LIN {X 0,Y 509.842,Z 166.475,A -85,B 0,C 180,E1 -5630.648,E2 -5630.648} C_VEL
LIN {X 0,Y 509.826,Z 166.476,A -85,B 0,C 180,E1 -5633.734,E2 -5633.734} C_VEL
LIN {X 0,Y 509.16,Z 166.561,A -85,B 0,C 180,E1 -5634.394,E2 -5634.394} C_VEL
LIN {X 0,Y 506.343,Z 166.91,A -85,B 0,C 180,E1 -5635.466,E2 -5635.466} C_VEL
LIN {X 0,Y 503.95,Z 167.21,A -85,B 0,C 180,E1 -5636.329,E2 -5636.329} C_VEL
LIN {X 0,Y 502.902,Z 167.337,A -85,B 0,C 180,E1 -5636.996,E2 -5636.996} C_VEL
LIN {X 0,Y 502.805,Z 167.349,A -85,B 0,C 180,E1 -5637.221,E2 -5637.221} C_VEL
LIN {X 0,Y 502.826,Z 167.352,A -85,B 0,C 180,E1 -5640.062,E2 -5640.062} C_VEL
LIN {X 0,Y 502.83,Z 167.346,A -85,B 0,C 180,E1 -5642.533,E2 -5642.533} C_VEL
LIN {X 0,Y 502.824,Z 167.349,A -85,B 0,C 180,E1 -5645.299,E2 -5645.299} C_VEL
LIN {X 0,Y 502.781,Z 167.358,A -85,B 0,C 180,E1 -5647.827,E2 -5647.827} C_VEL
LIN {X 0,Y 502.821,Z 167.347,A -85,B 0,C 180,E1 -5650.4,E2 -5650.4} C_VEL
LIN {X 0,Y 502.83,Z 167.349,A -85,B 0,C 180,E1 -5652.932,E2 -5652.932} C_VEL
LIN {X 0,Y 502.848,Z 167.352,A -85,B 0,C 180,E1 -5655.43,E2 -5655.43} C_VEL
LIN {X 0,Y 502.874,Z 167.343,A -85,B 0,C 180,E1 -5658.717,E2 -5658.717} C_VEL
LIN {X 0,Y 502.899,Z 167.34,A -85,B 0,C 180,E1 -5661.967,E2 -5661.967} C_VEL
LIN {X 0,Y 502.939,Z 167.335,A -85,B 0,C 180,E1 -5664.387,E2 -5664.387} C_VEL
LIN {X 0,Y 503.023,Z 167.326,A -85,B 0,C 180,E1 -5667.598,E2 -5667.598} C_VEL
LIN {X 0,Y 503.025,Z 167.324,A -85,B 0,C 180,E1 -5670,E2 -5670} C_VEL
LIN {X 0,Y 503.023,Z 167.326,A -85,B 0,C 180,E1 -5672.402,E2 -5672.402} C_VEL
LIN {X 0,Y 502.939,Z 167.335,A -85,B 0,C 180,E1 -5675.613,E2 -5675.613} C_VEL
LIN {X 0,Y 502.899,Z 167.34,A -85,B 0,C 180,E1 -5678.033,E2 -5678.033} C_VEL
LIN {X 0,Y 502.874,Z 167.343,A -85,B 0,C 180,E1 -5681.283,E2 -5681.283} C_VEL
LIN {X 0,Y 502.848,Z 167.352,A -85,B 0,C 180,E1 -5684.57,E2 -5684.57} C_VEL
LIN {X 0,Y 502.858,Z 167.346,A -85,B 0,C 180,E1 -5687.907,E2 -5687.907} C_VEL
LIN {X 0,Y 502.824,Z 167.353,A -85,B 0,C 180,E1 -5690.536,E2 -5690.536} C_VEL
LIN {X 0,Y 502.793,Z 167.351,A -85,B 0,C 180,E1 -5693.04,E2 -5693.04} C_VEL
LIN {X 0,Y 502.836,Z 167.346,A -85,B 0,C 180,E1 -5695.675,E2 -5695.675} C_VEL
LIN {X 0,Y 502.838,Z 167.35,A -85,B 0,C 180,E1 -5698.372,E2 -5698.372} C_VEL
LIN {X 0,Y 502.792,Z 167.352,A -85,B 0,C 180,E1 -5701.5,E2 -5701.5} C_VEL
LIN {X 0,Y 502.801,Z 167.352,A -85,B 0,C 180,E1 -5704.445,E2 -5704.445} C_VEL
LIN {X 0,Y 502.776,Z 167.353,A -85,B 0,C 180,E1 -5707.178,E2 -5707.178} C_VEL
LIN {X 0,Y 502.816,Z 167.353,A -85,B 0,C 180,E1 -5710.012,E2 -5710.012} C_VEL
LIN {X 0,Y 502.767,Z 167.356,A -85,B 0,C 180,E1 -5713.231,E2 -5713.231} C_VEL
LIN {X 0,Y 502.784,Z 167.36,A -85,B 0,C 180,E1 -5715.661,E2 -5715.661} C_VEL
LIN {X 0,Y 502.82,Z 167.349,A -85,B 0,C 180,E1 -5719.004,E2 -5719.004} C_VEL
LIN {X 0,Y 502.788,Z 167.352,A -85,B 0,C 180,E1 -5722.046,E2 -5722.046} C_VEL
LIN {X 0,Y 502.803,Z 167.353,A -85,B 0,C 180,E1 -5725.035,E2 -5725.035} C_VEL
LIN {X 0,Y 502.778,Z 167.353,A -85,B 0,C 180,E1 -5727.916,E2 -5727.916} C_VEL
LIN {X 0,Y 502.833,Z 167.348,A -85,B 0,C 180,E1 -5730.713,E2 -5730.713} C_VEL
LIN {X 0,Y 502.855,Z 167.346,A -85,B 0,C 180,E1 -5733.439,E2 -5733.439} C_VEL
LIN {X 0,Y 502.784,Z 167.351,A -85,B 0,C 180,E1 -5736.086,E2 -5736.086} C_VEL
LIN {X 0,Y 502.777,Z 167.357,A -85,B 0,C 180,E1 -5738.689,E2 -5738.689} C_VEL
LIN {X 0,Y 502.823,Z 167.35,A -85,B 0,C 180,E1 -5741.249,E2 -5741.249} C_VEL
LIN {X 0,Y 502.816,Z 167.347,A -85,B 0,C 180,E1 -5743.767,E2 -5743.767} C_VEL
LIN {X 0,Y 502.825,Z 167.349,A -85,B 0,C 180,E1 -5746.255,E2 -5746.255} C_VEL
LIN {X 0,Y 502.87,Z 167.348,A -85,B 0,C 180,E1 -5748.717,E2 -5748.717} C_VEL
LIN {X 0,Y 502.895,Z 167.339,A -85,B 0,C 180,E1 -5751.967,E2 -5751.967} C_VEL
LIN {X 0,Y 502.931,Z 167.34,A -85,B 0,C 180,E1 -5754.387,E2 -5754.387} C_VEL
LIN {X 0,Y 503.017,Z 167.323,A -85,B 0,C 180,E1 -5757.598,E2 -5757.598} C_VEL
LIN {X 0,Y 503.019,Z 167.326,A -85,B 0,C 180,E1 -5760,E2 -5760} C_VEL
LIN {X 0,Y 503.017,Z 167.329,A -85,B 0,C 180,E1 -5762.403,E2 -5762.403} C_VEL
LIN {X 0,Y 502.929,Z 167.335,A -85,B 0,C 180,E1 -5765.614,E2 -5765.614} C_VEL
LIN {X 0,Y 502.896,Z 167.346,A -85,B 0,C 180,E1 -5768.034,E2 -5768.034} C_VEL
LIN {X 0,Y 502.872,Z 167.341,A -85,B 0,C 180,E1 -5771.284,E2 -5771.284} C_VEL
LIN {X 0,Y 502.84,Z 167.345,A -85,B 0,C 180,E1 -5774.571,E2 -5774.571} C_VEL
LIN {X 0,Y 502.85,Z 167.35,A -85,B 0,C 180,E1 -5777.908,E2 -5777.908} C_VEL
LIN {X 0,Y 502.824,Z 167.346,A -85,B 0,C 180,E1 -5780.537,E2 -5780.537} C_VEL
LIN {X 0,Y 502.789,Z 167.352,A -85,B 0,C 180,E1 -5783.041,E2 -5783.041} C_VEL
LIN {X 0,Y 502.835,Z 167.352,A -85,B 0,C 180,E1 -5785.676,E2 -5785.676} C_VEL
LIN {X 0,Y 502.833,Z 167.345,A -85,B 0,C 180,E1 -5788.374,E2 -5788.374} C_VEL
LIN {X 0,Y 502.789,Z 167.357,A -85,B 0,C 180,E1 -5791.499,E2 -5791.499} C_VEL
LIN {X 0,Y 502.8,Z 167.352,A -85,B 0,C 180,E1 -5793.995,E2 -5793.995} C_VEL
LIN {X 0,Y 502.775,Z 167.361,A -85,B 0,C 180,E1 -5797.178,E2 -5797.178} C_VEL
LIN {X 0,Y 502.785,Z 167.355,A -85,B 0,C 180,E1 -5800.016,E2 -5800.016} C_VEL
LIN {X 0,Y 502.801,Z 167.354,A -85,B 0,C 180,E1 -5802.2,E2 -5802.2} C_VEL
LIN {X 0,Y 502.757,Z 167.362,A -85,B 0,C 180,E1 -5803.374,E2 -5803.374} C_VEL
LIN {X 0,Y 502.897,Z 168.072,A -85,B 0,C 180,E1 -5804.544,E2 -5804.544} C_VEL
LIN {X 0,Y 503.501,Z 172.327,A -85,B 0,C 180,E1 -5807.714,E2 -5807.714} C_VEL
LIN {X 0,Y 503.568,Z 175.925,A -85,B 0,C 180,E1 -5810.14,E2 -5810.14} C_VEL
LIN {X 0,Y 503.28,Z 180.665,A -85,B 0,C 180,E1 -5813.097,E2 -5813.097} C_VEL
LIN {X 0,Y 503.059,Z 185.701,A -85,B 0,C 180,E1 -5816.026,E2 -5816.026} C_VEL
LIN {X 0,Y 502.876,Z 190.836,A -85,B 0,C 180,E1 -5818.863,E2 -5818.863} C_VEL
LIN {X 0,Y 502.695,Z 196.322,A -85,B 0,C 180,E1 -5821.737,E2 -5821.737} C_VEL
LIN {X 0,Y 502.576,Z 201.398,A -85,B 0,C 180,E1 -5824.31,E2 -5824.31} C_VEL
LIN {X 0,Y 502.48,Z 207.799,A -85,B 0,C 180,E1 -5827.387,E2 -5827.387} C_VEL
LIN {X 0,Y 502.354,Z 214.071,A -85,B 0,C 180,E1 -5830.381,E2 -5830.381} C_VEL
LIN {X 0,Y 502.241,Z 219.461,A -85,B 0,C 180,E1 -5832.911,E2 -5832.911} C_VEL
LIN {X 0,Y 502.211,Z 225.524,A -85,B 0,C 180,E1 -5835.721,E2 -5835.721} C_VEL
LIN {X 0,Y 504.275,Z 237.727,A -85,B 0,C 180,E1 -5836.089,E2 -5836.089} C_VEL
LIN {X 0,Y 504.627,Z 241.055,A -85,B 0,C 180,E1 -5836.202,E2 -5836.202} C_VEL
LIN {X 0,Y 504.312,Z 253.379,A -85,B 0,C 180,E1 -5836.707,E2 -5836.707} C_VEL
LIN {X 0,Y 504.006,Z 263.916,A -85,B 0,C 180,E1 -5837.276,E2 -5837.276} C_VEL
LIN {X 0,Y 503.684,Z 273.477,A -85,B 0,C 180,E1 -5837.919,E2 -5837.919} C_VEL
LIN {X 0,Y 503.425,Z 282.175,A -85,B 0,C 180,E1 -5838.627,E2 -5838.627} C_VEL
LIN {X 0,Y 503.194,Z 289.542,A -85,B 0,C 180,E1 -5839.336,E2 -5839.336} C_VEL
LIN {X 0,Y 502.944,Z 296.73,A -85,B 0,C 180,E1 -5840.144,E2 -5840.144} C_VEL
LIN {X 0,Y 502.683,Z 304.275,A -85,B 0,C 180,E1 -5841.153,E2 -5841.153} C_VEL
LIN {X 0,Y 502.471,Z 310.565,A -85,B 0,C 180,E1 -5842.162,E2 -5842.162} C_VEL
LIN {X 0,Y 502.317,Z 315.989,A -85,B 0,C 180,E1 -5843.21,E2 -5843.21} C_VEL
LIN {X 0,Y 502.256,Z 320.895,A -85,B 0,C 180,E1 -5844.379,E2 -5844.379} C_VEL
LIN {X 0,Y 502.128,Z 324.85,A -85,B 0,C 180,E1 -5845.585,E2 -5845.585} C_VEL
LIN {X 0,Y 502.122,Z 327.772,A -85,B 0,C 180,E1 -5846.791,E2 -5846.791} C_VEL
LIN {X 0,Y 502.036,Z 330.196,A -85,B 0,C 180,E1 -5848.396,E2 -5848.396} C_VEL
LIN {X 0,Y 501.99,Z 330.78,A -85,B 0,C 180,E1 -5849.198,E2 -5849.198} C_VEL
LIN {X 0,Y 501.99,Z 330.78,A -85,B 0,C 180,E1 -5850.802,E2 -5850.802} C_VEL
LIN {X 0,Y 502.036,Z 330.196,A -85,B 0,C 180,E1 -5851.604,E2 -5851.604} C_VEL
LIN {X 0,Y 502.122,Z 327.772,A -85,B 0,C 180,E1 -5853.209,E2 -5853.209} C_VEL
LIN {X 0,Y 502.128,Z 324.85,A -85,B 0,C 180,E1 -5854.415,E2 -5854.415} C_VEL
LIN {X 0,Y 502.257,Z 320.895,A -85,B 0,C 180,E1 -5855.621,E2 -5855.621} C_VEL
LIN {X 0,Y 502.317,Z 315.989,A -85,B 0,C 180,E1 -5856.79,E2 -5856.79} C_VEL
LIN {X 0,Y 502.471,Z 310.565,A -85,B 0,C 180,E1 -5857.838,E2 -5857.838} C_VEL
LIN {X 0,Y 502.683,Z 304.275,A -85,B 0,C 180,E1 -5858.847,E2 -5858.847} C_VEL
LIN {X 0,Y 502.944,Z 296.73,A -85,B 0,C 180,E1 -5859.856,E2 -5859.856} C_VEL
LIN {X 0,Y 503.237,Z 287.621,A -85,B 0,C 180,E1 -5860.867,E2 -5860.867} C_VEL
LIN {X 0,Y 503.648,Z 276.174,A -85,B 0,C 180,E1 -5861.878,E2 -5861.878} C_VEL
LIN {X 0,Y 503.876,Z 266.59,A -85,B 0,C 180,E1 -5862.559,E2 -5862.559} C_VEL
LIN {X 0,Y 504.174,Z 256.395,A -85,B 0,C 180,E1 -5863.143,E2 -5863.143} C_VEL
LIN {X 0,Y 504.477,Z 246.331,A -85,B 0,C 180,E1 -5863.597,E2 -5863.597} C_VEL
LIN {X 0,Y 504.441,Z 238.601,A -85,B 0,C 180,E1 -5863.88,E2 -5863.88} C_VEL
LIN {X 0,Y 502.532,Z 227.434,A -85,B 0,C 180,E1 -5864.227,E2 -5864.227} C_VEL
LIN {X 0,Y 502.211,Z 225.524,A -85,B 0,C 180,E1 -5864.279,E2 -5864.279} C_VEL
LIN {X 0,Y 502.241,Z 219.461,A -85,B 0,C 180,E1 -5867.089,E2 -5867.089} C_VEL
LIN {X 0,Y 502.421,Z 212.275,A -85,B 0,C 180,E1 -5870.469,E2 -5870.469} C_VEL
LIN {X 0,Y 502.479,Z 206.885,A -85,B 0,C 180,E1 -5873.055,E2 -5873.055} C_VEL
LIN {X 0,Y 502.576,Z 201.398,A -85,B 0,C 180,E1 -5875.69,E2 -5875.69} C_VEL
LIN {X 0,Y 502.702,Z 196.094,A -85,B 0,C 180,E1 -5878.381,E2 -5878.381} C_VEL
LIN {X 0,Y 502.876,Z 190.832,A -85,B 0,C 180,E1 -5881.137,E2 -5881.137} C_VEL
LIN {X 0,Y 503.052,Z 185.669,A -85,B 0,C 180,E1 -5883.974,E2 -5883.974} C_VEL
LIN {X 0,Y 503.329,Z 180.065,A -85,B 0,C 180,E1 -5887.26,E2 -5887.26} C_VEL
LIN {X 0,Y 503.544,Z 175.787,A -85,B 0,C 180,E1 -5889.942,E2 -5889.942} C_VEL
LIN {X 0,Y 503.509,Z 172.318,A -85,B 0,C 180,E1 -5892.287,E2 -5892.287} C_VEL
LIN {X 0,Y 502.897,Z 168.091,A -85,B 0,C 180,E1 -5895.456,E2 -5895.456} C_VEL
LIN {X 0,Y 502.755,Z 167.361,A -85,B 0,C 180,E1 -5896.766,E2 -5896.766} C_VEL
LIN {X 0,Y 502.796,Z 167.358,A -85,B 0,C 180,E1 -5899.007,E2 -5899.007} C_VEL
LIN {X 0,Y 502.79,Z 167.354,A -85,B 0,C 180,E1 -5902.045,E2 -5902.045} C_VEL
LIN {X 0,Y 502.795,Z 167.357,A -85,B 0,C 180,E1 -5905.033,E2 -5905.033} C_VEL
LIN {X 0,Y 502.78,Z 167.352,A -85,B 0,C 180,E1 -5907.915,E2 -5907.915} C_VEL
LIN {X 0,Y 502.818,Z 167.353,A -85,B 0,C 180,E1 -5910.711,E2 -5910.711} C_VEL
LIN {X 0,Y 502.859,Z 167.342,A -85,B 0,C 180,E1 -5913.439,E2 -5913.439} C_VEL
LIN {X 0,Y 502.787,Z 167.355,A -85,B 0,C 180,E1 -5916.086,E2 -5916.086} C_VEL
LIN {X 0,Y 502.779,Z 167.355,A -85,B 0,C 180,E1 -5918.688,E2 -5918.688} C_VEL
LIN {X 0,Y 502.824,Z 167.346,A -85,B 0,C 180,E1 -5921.248,E2 -5921.248} C_VEL
LIN {X 0,Y 502.816,Z 167.35,A -85,B 0,C 180,E1 -5923.767,E2 -5923.767} C_VEL
LIN {X 0,Y 502.825,Z 167.352,A -85,B 0,C 180,E1 -5926.254,E2 -5926.254} C_VEL
LIN {X 0,Y 502.872,Z 167.341,A -85,B 0,C 180,E1 -5928.716,E2 -5928.716} C_VEL
LIN {X 0,Y 502.896,Z 167.346,A -85,B 0,C 180,E1 -5931.966,E2 -5931.966} C_VEL
LIN {X 0,Y 502.929,Z 167.335,A -85,B 0,C 180,E1 -5934.386,E2 -5934.386} C_VEL
LIN {X 0,Y 503.017,Z 167.329,A -85,B 0,C 180,E1 -5937.597,E2 -5937.597} C_VEL
LIN {X 0,Y 503.019,Z 167.326,A -85,B 0,C 180,E1 -5940,E2 -5940} C_VEL
LIN {X 0,Y 503.017,Z 167.323,A -85,B 0,C 180,E1 -5942.402,E2 -5942.402} C_VEL
LIN {X 0,Y 502.931,Z 167.34,A -85,B 0,C 180,E1 -5945.613,E2 -5945.613} C_VEL
LIN {X 0,Y 502.895,Z 167.339,A -85,B 0,C 180,E1 -5948.033,E2 -5948.033} C_VEL
LIN {X 0,Y 502.87,Z 167.348,A -85,B 0,C 180,E1 -5951.283,E2 -5951.283} C_VEL
LIN {X 0,Y 502.838,Z 167.345,A -85,B 0,C 180,E1 -5954.571,E2 -5954.571} C_VEL
LIN {X 0,Y 502.855,Z 167.343,A -85,B 0,C 180,E1 -5957.907,E2 -5957.907} C_VEL
LIN {X 0,Y 502.822,Z 167.348,A -85,B 0,C 180,E1 -5960.536,E2 -5960.536} C_VEL
LIN {X 0,Y 502.787,Z 167.359,A -85,B 0,C 180,E1 -5963.04,E2 -5963.04} C_VEL
LIN {X 0,Y 502.833,Z 167.346,A -85,B 0,C 180,E1 -5965.675,E2 -5965.675} C_VEL
LIN {X 0,Y 502.836,Z 167.347,A -85,B 0,C 180,E1 -5968.372,E2 -5968.372} C_VEL
LIN {X 0,Y 502.787,Z 167.351,A -85,B 0,C 180,E1 -5971.499,E2 -5971.499} C_VEL
LIN {X 0,Y 502.8,Z 167.355,A -85,B 0,C 180,E1 -5974.445,E2 -5974.445} C_VEL
LIN {X 0,Y 502.774,Z 167.354,A -85,B 0,C 180,E1 -5977.178,E2 -5977.178} C_VEL
LIN {X 0,Y 502.815,Z 167.35,A -85,B 0,C 180,E1 -5980.012,E2 -5980.012} C_VEL
LIN {X 0,Y 502.767,Z 167.354,A -85,B 0,C 180,E1 -5983.231,E2 -5983.231} C_VEL
LIN {X 0,Y 502.783,Z 167.352,A -85,B 0,C 180,E1 -5985.661,E2 -5985.661} C_VEL
LIN {X 0,Y 502.813,Z 167.348,A -85,B 0,C 180,E1 -5989.005,E2 -5989.005} C_VEL
LIN {X 0,Y 502.789,Z 167.358,A -85,B 0,C 180,E1 -5992.046,E2 -5992.046} C_VEL
LIN {X 0,Y 502.805,Z 167.349,A -85,B 0,C 180,E1 -5995.035,E2 -5995.035} C_VEL
LIN {X 0,Y 502.805,Z 167.349,A -85,B 0,C 180,E1 -5997.221,E2 -5997.221} C_VEL
LIN {X 0,Y 502.107,Z 167.443,A -85,B 0,C 180,E1 -5997.89,E2 -5997.89} C_VEL
LIN {X 0,Y 499.249,Z 167.796,A -85,B 0,C 180,E1 -5998.976,E2 -5998.976} C_VEL
LIN {X 0,Y 496.858,Z 168.098,A -85,B 0,C 180,E1 -5999.851,E2 -5999.851} C_VEL
LIN {X 0,Y 495.84,Z 168.218,A -85,B 0,C 180,E1 -6000.526,E2 -6000.526} C_VEL
LIN {X 0,Y 495.76,Z 168.226,A -85,B 0,C 180,E1 -6000.755,E2 -6000.755} C_VEL
LIN {X 0,Y 495.787,Z 168.229,A -85,B 0,C 180,E1 -6003.932,E2 -6003.932} C_VEL
LIN {X 0,Y 495.761,Z 168.228,A -85,B 0,C 180,E1 -6007.138,E2 -6007.138} C_VEL
LIN {X 0,Y 495.774,Z 168.227,A -85,B 0,C 180,E1 -6010.11,E2 -6010.11} C_VEL
LIN {X 0,Y 495.783,Z 168.226,A -85,B 0,C 180,E1 -6012.682,E2 -6012.682} C_VEL
LIN {X 0,Y 495.791,Z 168.23,A -85,B 0,C 180,E1 -6015.217,E2 -6015.217} C_VEL
LIN {X 0,Y 495.848,Z 168.218,A -85,B 0,C 180,E1 -6018.555,E2 -6018.555} C_VEL
LIN {X 0,Y 495.87,Z 168.217,A -85,B 0,C 180,E1 -6021.852,E2 -6021.852} C_VEL
LIN {X 0,Y 495.896,Z 168.212,A -85,B 0,C 180,E1 -6024.307,E2 -6024.307} C_VEL
LIN {X 0,Y 495.991,Z 168.202,A -85,B 0,C 180,E1 -6027.564,E2 -6027.564} C_VEL
LIN {X 0,Y 495.996,Z 168.2,A -85,B 0,C 180,E1 -6030,E2 -6030} C_VEL
LIN {X 0,Y 495.992,Z 168.202,A -85,B 0,C 180,E1 -6032.436,E2 -6032.436} C_VEL
LIN {X 0,Y 495.896,Z 168.212,A -85,B 0,C 180,E1 -6035.693,E2 -6035.693} C_VEL
LIN {X 0,Y 495.87,Z 168.217,A -85,B 0,C 180,E1 -6038.148,E2 -6038.148} C_VEL
LIN {X 0,Y 495.848,Z 168.218,A -85,B 0,C 180,E1 -6041.445,E2 -6041.445} C_VEL
LIN {X 0,Y 495.791,Z 168.23,A -85,B 0,C 180,E1 -6044.783,E2 -6044.783} C_VEL
LIN {X 0,Y 495.783,Z 168.226,A -85,B 0,C 180,E1 -6047.318,E2 -6047.318} C_VEL
LIN {X 0,Y 495.774,Z 168.227,A -85,B 0,C 180,E1 -6049.89,E2 -6049.89} C_VEL
LIN {X 0,Y 495.761,Z 168.228,A -85,B 0,C 180,E1 -6052.862,E2 -6052.862} C_VEL
LIN {X 0,Y 495.787,Z 168.229,A -85,B 0,C 180,E1 -6056.068,E2 -6056.068} C_VEL
LIN {X 0,Y 495.776,Z 168.225,A -85,B 0,C 180,E1 -6058.814,E2 -6058.814} C_VEL
LIN {X 0,Y 495.755,Z 168.231,A -85,B 0,C 180,E1 -6061.726,E2 -6061.726} C_VEL
LIN {X 0,Y 495.771,Z 168.225,A -85,B 0,C 180,E1 -6064.695,E2 -6064.695} C_VEL
LIN {X 0,Y 495.726,Z 168.235,A -85,B 0,C 180,E1 -6067.561,E2 -6067.561} C_VEL
LIN {X 0,Y 495.774,Z 168.225,A -85,B 0,C 180,E1 -6070.698,E2 -6070.698} C_VEL
LIN {X 0,Y 495.727,Z 168.234,A -85,B 0,C 180,E1 -6074.001,E2 -6074.001} C_VEL
LIN {X 0,Y 495.719,Z 168.234,A -85,B 0,C 180,E1 -6077.117,E2 -6077.117} C_VEL
LIN {X 0,Y 495.783,Z 168.226,A -85,B 0,C 180,E1 -6079.949,E2 -6079.949} C_VEL
LIN {X 0,Y 495.724,Z 168.231,A -85,B 0,C 180,E1 -6082.553,E2 -6082.553} C_VEL
LIN {X 0,Y 495.778,Z 168.231,A -85,B 0,C 180,E1 -6085.457,E2 -6085.457} C_VEL
LIN {X 0,Y 495.75,Z 168.228,A -85,B 0,C 180,E1 -6088.364,E2 -6088.364} C_VEL
LIN {X 0,Y 495.783,Z 168.227,A -85,B 0,C 180,E1 -6091.506,E2 -6091.506} C_VEL
LIN {X 0,Y 495.784,Z 168.224,A -85,B 0,C 180,E1 -6093.932,E2 -6093.932} C_VEL
LIN {X 0,Y 495.754,Z 168.233,A -85,B 0,C 180,E1 -6097.139,E2 -6097.139} C_VEL
LIN {X 0,Y 495.771,Z 168.225,A -85,B 0,C 180,E1 -6100.11,E2 -6100.11} C_VEL
LIN {X 0,Y 495.78,Z 168.23,A -85,B 0,C 180,E1 -6102.682,E2 -6102.682} C_VEL
LIN {X 0,Y 495.783,Z 168.226,A -85,B 0,C 180,E1 -6105.217,E2 -6105.217} C_VEL
LIN {X 0,Y 495.845,Z 168.223,A -85,B 0,C 180,E1 -6108.555,E2 -6108.555} C_VEL
LIN {X 0,Y 495.867,Z 168.214,A -85,B 0,C 180,E1 -6111.852,E2 -6111.852} C_VEL
LIN {X 0,Y 495.889,Z 168.216,A -85,B 0,C 180,E1 -6114.307,E2 -6114.307} C_VEL
LIN {X 0,Y 495.986,Z 168.198,A -85,B 0,C 180,E1 -6117.564,E2 -6117.564} C_VEL
LIN {X 0,Y 495.991,Z 168.202,A -85,B 0,C 180,E1 -6120,E2 -6120} C_VEL
LIN {X 0,Y 495.986,Z 168.204,A -85,B 0,C 180,E1 -6122.437,E2 -6122.437} C_VEL
LIN {X 0,Y 495.885,Z 168.213,A -85,B 0,C 180,E1 -6125.694,E2 -6125.694} C_VEL
LIN {X 0,Y 495.867,Z 168.22,A -85,B 0,C 180,E1 -6128.148,E2 -6128.148} C_VEL
LIN {X 0,Y 495.846,Z 168.217,A -85,B 0,C 180,E1 -6131.446,E2 -6131.446} C_VEL
LIN {X 0,Y 495.785,Z 168.223,A -85,B 0,C 180,E1 -6134.783,E2 -6134.783} C_VEL
LIN {X 0,Y 495.776,Z 168.227,A -85,B 0,C 180,E1 -6137.319,E2 -6137.319} C_VEL
LIN {X 0,Y 495.767,Z 168.232,A -85,B 0,C 180,E1 -6139.891,E2 -6139.891} C_VEL
LIN {X 0,Y 495.757,Z 168.227,A -85,B 0,C 180,E1 -6142.862,E2 -6142.862} C_VEL
LIN {X 0,Y 495.786,Z 168.225,A -85,B 0,C 180,E1 -6146.069,E2 -6146.069} C_VEL
LIN {X 0,Y 495.765,Z 168.227,A -85,B 0,C 180,E1 -6148.816,E2 -6148.816} C_VEL
LIN {X 0,Y 495.752,Z 168.231,A -85,B 0,C 180,E1 -6151.726,E2 -6151.726} C_VEL
LIN {X 0,Y 495.765,Z 168.229,A -85,B 0,C 180,E1 -6154.695,E2 -6154.695} C_VEL
LIN {X 0,Y 495.726,Z 168.237,A -85,B 0,C 180,E1 -6157.562,E2 -6157.562} C_VEL
LIN {X 0,Y 495.756,Z 168.231,A -85,B 0,C 180,E1 -6160.048,E2 -6160.048} C_VEL
LIN {X 0,Y 495.715,Z 168.24,A -85,B 0,C 180,E1 -6162.885,E2 -6162.885} C_VEL
LIN {X 0,Y 495.736,Z 168.3,A -85,B 0,C 180,E1 -6163.696,E2 -6163.696} C_VEL
LIN {X 0,Y 496.228,Z 171.553,A -85,B 0,C 180,E1 -6166.246,E2 -6166.246} C_VEL
LIN {X 0,Y 496.573,Z 174.792,A -85,B 0,C 180,E1 -6168.6,E2 -6168.6} C_VEL
LIN {X 0,Y 496.474,Z 178.608,A -85,B 0,C 180,E1 -6171.13,E2 -6171.13} C_VEL
LIN {X 0,Y 496.21,Z 182.969,A -85,B 0,C 180,E1 -6173.835,E2 -6173.835} C_VEL
LIN {X 0,Y 495.978,Z 187.922,A -85,B 0,C 180,E1 -6176.724,E2 -6176.724} C_VEL
LIN {X 0,Y 495.784,Z 193.591,A -85,B 0,C 180,E1 -6179.85,E2 -6179.85} C_VEL
LIN {X 0,Y 495.608,Z 200.151,A -85,B 0,C 180,E1 -6183.301,E2 -6183.301} C_VEL
LIN {X 0,Y 495.463,Z 204.973,A -85,B 0,C 180,E1 -6185.71,E2 -6185.71} C_VEL
LIN {X 0,Y 495.381,Z 210.478,A -85,B 0,C 180,E1 -6188.355,E2 -6188.355} C_VEL
LIN {X 0,Y 495.244,Z 215.868,A -85,B 0,C 180,E1 -6190.95,E2 -6190.95} C_VEL
LIN {X 0,Y 495.137,Z 221.257,A -85,B 0,C 180,E1 -6193.508,E2 -6193.508} C_VEL
LIN {X 0,Y 495.124,Z 225.524,A -85,B 0,C 180,E1 -6195.512,E2 -6195.512} C_VEL
LIN {X 0,Y 497.25,Z 237.711,A -85,B 0,C 180,E1 -6195.889,E2 -6195.889} C_VEL
LIN {X 0,Y 497.752,Z 241.06,A -85,B 0,C 180,E1 -6196.008,E2 -6196.008} C_VEL
LIN {X 0,Y 497.407,Z 253.37,A -85,B 0,C 180,E1 -6196.519,E2 -6196.519} C_VEL
LIN {X 0,Y 497.05,Z 264.161,A -85,B 0,C 180,E1 -6197.111,E2 -6197.111} C_VEL
LIN {X 0,Y 496.736,Z 273.469,A -85,B 0,C 180,E1 -6197.747,E2 -6197.747} C_VEL
LIN {X 0,Y 496.433,Z 282.169,A -85,B 0,C 180,E1 -6198.465,E2 -6198.465} C_VEL
LIN {X 0,Y 496.203,Z 289.536,A -85,B 0,C 180,E1 -6199.184,E2 -6199.184} C_VEL
LIN {X 0,Y 495.924,Z 296.726,A -85,B 0,C 180,E1 -6200.003,E2 -6200.003} C_VEL
LIN {X 0,Y 495.634,Z 304.271,A -85,B 0,C 180,E1 -6201.027,E2 -6201.027} C_VEL
LIN {X 0,Y 495.403,Z 310.56,A -85,B 0,C 180,E1 -6202.05,E2 -6202.05} C_VEL
LIN {X 0,Y 495.247,Z 315.984,A -85,B 0,C 180,E1 -6203.113,E2 -6203.113} C_VEL
LIN {X 0,Y 495.174,Z 320.891,A -85,B 0,C 180,E1 -6204.298,E2 -6204.298} C_VEL
LIN {X 0,Y 495.029,Z 324.847,A -85,B 0,C 180,E1 -6205.522,E2 -6205.522} C_VEL
LIN {X 0,Y 495.045,Z 327.769,A -85,B 0,C 180,E1 -6206.745,E2 -6206.745} C_VEL
LIN {X 0,Y 494.961,Z 330.195,A -85,B 0,C 180,E1 -6208.373,E2 -6208.373} C_VEL
LIN {X 0,Y 494.911,Z 330.779,A -85,B 0,C 180,E1 -6209.186,E2 -6209.186} C_VEL
LIN {X 0,Y 494.911,Z 330.779,A -85,B 0,C 180,E1 -6210.814,E2 -6210.814} C_VEL
LIN {X 0,Y 494.961,Z 330.195,A -85,B 0,C 180,E1 -6211.627,E2 -6211.627} C_VEL
LIN {X 0,Y 495.045,Z 327.769,A -85,B 0,C 180,E1 -6213.255,E2 -6213.255} C_VEL
LIN {X 0,Y 495.029,Z 324.847,A -85,B 0,C 180,E1 -6214.478,E2 -6214.478} C_VEL
LIN {X 0,Y 495.175,Z 320.891,A -85,B 0,C 180,E1 -6215.702,E2 -6215.702} C_VEL
LIN {X 0,Y 495.247,Z 315.984,A -85,B 0,C 180,E1 -6216.887,E2 -6216.887} C_VEL
LIN {X 0,Y 495.403,Z 310.56,A -85,B 0,C 180,E1 -6217.95,E2 -6217.95} C_VEL
LIN {X 0,Y 495.634,Z 304.271,A -85,B 0,C 180,E1 -6218.973,E2 -6218.973} C_VEL
LIN {X 0,Y 495.925,Z 296.726,A -85,B 0,C 180,E1 -6219.997,E2 -6219.997} C_VEL
LIN {X 0,Y 496.226,Z 287.618,A -85,B 0,C 180,E1 -6221.023,E2 -6221.023} C_VEL
LIN {X 0,Y 496.688,Z 276.166,A -85,B 0,C 180,E1 -6222.046,E2 -6222.046} C_VEL
LIN {X 0,Y 496.916,Z 267.071,A -85,B 0,C 180,E1 -6222.707,E2 -6222.707} C_VEL
LIN {X 0,Y 497.24,Z 256.386,A -85,B 0,C 180,E1 -6223.33,E2 -6223.33} C_VEL
LIN {X 0,Y 497.576,Z 246.321,A -85,B 0,C 180,E1 -6223.789,E2 -6223.789} C_VEL
LIN {X 0,Y 497.529,Z 239.458,A -85,B 0,C 180,E1 -6224.051,E2 -6224.051} C_VEL
LIN {X 0,Y 495.381,Z 227.148,A -85,B 0,C 180,E1 -6224.442,E2 -6224.442} C_VEL
LIN {X 0,Y 495.124,Z 225.524,A -85,B 0,C 180,E1 -6224.488,E2 -6224.488} C_VEL
LIN {X 0,Y 495.217,Z 217.99,A -85,B 0,C 180,E1 -6228.038,E2 -6228.038} C_VEL
LIN {X 0,Y 495.341,Z 212.275,A -85,B 0,C 180,E1 -6230.775,E2 -6230.775} C_VEL
LIN {X 0,Y 495.429,Z 206.812,A -85,B 0,C 180,E1 -6233.403,E2 -6233.403} C_VEL
LIN {X 0,Y 495.537,Z 201.352,A -85,B 0,C 180,E1 -6236.082,E2 -6236.082} C_VEL
LIN {X 0,Y 495.676,Z 196.09,A -85,B 0,C 180,E1 -6238.82,E2 -6238.82} C_VEL
LIN {X 0,Y 495.867,Z 190.623,A -85,B 0,C 180,E1 -6241.745,E2 -6241.745} C_VEL
LIN {X 0,Y 496.076,Z 185.359,A -85,B 0,C 180,E1 -6244.744,E2 -6244.744} C_VEL
LIN {X 0,Y 496.331,Z 180.7,A -85,B 0,C 180,E1 -6247.537,E2 -6247.537} C_VEL
LIN {X 0,Y 496.534,Z 176.625,A -85,B 0,C 180,E1 -6250.153,E2 -6250.153} C_VEL
LIN {X 0,Y 496.579,Z 174.356,A -85,B 0,C 180,E1 -6251.696,E2 -6251.696} C_VEL
LIN {X 0,Y 496.17,Z 171.277,A -85,B 0,C 180,E1 -6253.951,E2 -6253.951} C_VEL
LIN {X 0,Y 495.736,Z 168.296,A -85,B 0,C 180,E1 -6256.304,E2 -6256.304} C_VEL
LIN {X 0,Y 495.751,Z 168.234,A -85,B 0,C 180,E1 -6259.298,E2 -6259.298} C_VEL
LIN {X 0,Y 495.748,Z 168.233,A -85,B 0,C 180,E1 -6261.408,E2 -6261.408} C_VEL
LIN {X 0,Y 495.745,Z 168.233,A -85,B 0,C 180,E1 -6264.462,E2 -6264.462} C_VEL
LIN {X 0,Y 495.764,Z 168.226,A -85,B 0,C 180,E1 -6267.405,E2 -6267.405} C_VEL
LIN {X 0,Y 495.762,Z 168.23,A -85,B 0,C 180,E1 -6270.253,E2 -6270.253} C_VEL
LIN {X 0,Y 495.819,Z 168.219,A -85,B 0,C 180,E1 -6273.25,E2 -6273.25} C_VEL
LIN {X 0,Y 495.748,Z 168.229,A -85,B 0,C 180,E1 -6275.724,E2 -6275.724} C_VEL
LIN {X 0,Y 495.738,Z 168.237,A -85,B 0,C 180,E1 -6278.37,E2 -6278.37} C_VEL
LIN {X 0,Y 495.779,Z 168.225,A -85,B 0,C 180,E1 -6280.971,E2 -6280.971} C_VEL
LIN {X 0,Y 495.773,Z 168.226,A -85,B 0,C 180,E1 -6283.529,E2 -6283.529} C_VEL
LIN {X 0,Y 495.788,Z 168.231,A -85,B 0,C 180,E1 -6286.055,E2 -6286.055} C_VEL
LIN {X 0,Y 495.846,Z 168.217,A -85,B 0,C 180,E1 -6288.554,E2 -6288.554} C_VEL
LIN {X 0,Y 495.867,Z 168.22,A -85,B 0,C 180,E1 -6291.852,E2 -6291.852} C_VEL
LIN {X 0,Y 495.885,Z 168.213,A -85,B 0,C 180,E1 -6294.306,E2 -6294.306} C_VEL
LIN {X 0,Y 495.986,Z 168.204,A -85,B 0,C 180,E1 -6297.563,E2 -6297.563} C_VEL
LIN {X 0,Y 495.991,Z 168.202,A -85,B 0,C 180,E1 -6300,E2 -6300} C_VEL
LIN {X 0,Y 495.986,Z 168.198,A -85,B 0,C 180,E1 -6302.436,E2 -6302.436} C_VEL
LIN {X 0,Y 495.889,Z 168.216,A -85,B 0,C 180,E1 -6305.693,E2 -6305.693} C_VEL
LIN {X 0,Y 495.867,Z 168.214,A -85,B 0,C 180,E1 -6308.148,E2 -6308.148} C_VEL
LIN {X 0,Y 495.845,Z 168.223,A -85,B 0,C 180,E1 -6311.445,E2 -6311.445} C_VEL
LIN {X 0,Y 495.783,Z 168.226,A -85,B 0,C 180,E1 -6314.783,E2 -6314.783} C_VEL
LIN {X 0,Y 495.78,Z 168.23,A -85,B 0,C 180,E1 -6317.318,E2 -6317.318} C_VEL
LIN {X 0,Y 495.771,Z 168.225,A -85,B 0,C 180,E1 -6319.89,E2 -6319.89} C_VEL
LIN {X 0,Y 495.754,Z 168.233,A -85,B 0,C 180,E1 -6322.861,E2 -6322.861} C_VEL
LIN {X 0,Y 495.784,Z 168.224,A -85,B 0,C 180,E1 -6326.068,E2 -6326.068} C_VEL
LIN {X 0,Y 495.774,Z 168.233,A -85,B 0,C 180,E1 -6328.814,E2 -6328.814} C_VEL
LIN {X 0,Y 495.75,Z 168.228,A -85,B 0,C 180,E1 -6331.726,E2 -6331.726} C_VEL
LIN {X 0,Y 495.77,Z 168.233,A -85,B 0,C 180,E1 -6334.695,E2 -6334.695} C_VEL
LIN {X 0,Y 495.725,Z 168.231,A -85,B 0,C 180,E1 -6337.561,E2 -6337.561} C_VEL
LIN {X 0,Y 495.773,Z 168.23,A -85,B 0,C 180,E1 -6340.699,E2 -6340.699} C_VEL
LIN {X 0,Y 495.728,Z 168.234,A -85,B 0,C 180,E1 -6344.001,E2 -6344.001} C_VEL
LIN {X 0,Y 495.719,Z 168.232,A -85,B 0,C 180,E1 -6347.117,E2 -6347.117} C_VEL
LIN {X 0,Y 495.753,Z 168.232,A -85,B 0,C 180,E1 -6349.953,E2 -6349.953} C_VEL
LIN {X 0,Y 495.725,Z 168.233,A -85,B 0,C 180,E1 -6352.553,E2 -6352.553} C_VEL
LIN {X 0,Y 495.78,Z 168.225,A -85,B 0,C 180,E1 -6355.458,E2 -6355.458} C_VEL
LIN {X 0,Y 495.755,Z 168.23,A -85,B 0,C 180,E1 -6358.364,E2 -6358.364} C_VEL
LIN {X 0,Y 495.76,Z 168.226,A -85,B 0,C 180,E1 -6360.755,E2 -6360.755} C_VEL
LIN {X 0,Y 495.098,Z 168.313,A -85,B 0,C 180,E1 -6361.434,E2 -6361.434} C_VEL
LIN {X 0,Y 492.237,Z 168.666,A -85,B 0,C 180,E1 -6362.537,E2 -6362.537} C_VEL
LIN {X 0,Y 489.827,Z 168.969,A -85,B 0,C 180,E1 -6363.425,E2 -6363.425} C_VEL
LIN {X 0,Y 488.811,Z 169.096,A -85,B 0,C 180,E1 -6364.111,E2 -6364.111} C_VEL
LIN {X 0,Y 488.738,Z 169.102,A -85,B 0,C 180,E1 -6364.344,E2 -6364.344} C_VEL
LIN {X 0,Y 488.724,Z 169.105,A -85,B 0,C 180,E1 -6367.154,E2 -6367.154} C_VEL
LIN {X 0,Y 488.725,Z 169.11,A -85,B 0,C 180,E1 -6369.811,E2 -6369.811} C_VEL
LIN {X 0,Y 488.73,Z 169.105,A -85,B 0,C 180,E1 -6372.424,E2 -6372.424} C_VEL
LIN {X 0,Y 488.761,Z 169.103,A -85,B 0,C 180,E1 -6375,E2 -6375} C_VEL
LIN {X 0,Y 488.802,Z 169.095,A -85,B 0,C 180,E1 -6378.388,E2 -6378.388} C_VEL
LIN {X 0,Y 488.815,Z 169.097,A -85,B 0,C 180,E1 -6381.734,E2 -6381.734} C_VEL
LIN {X 0,Y 488.856,Z 169.089,A -85,B 0,C 180,E1 -6384.224,E2 -6384.224} C_VEL
LIN {X 0,Y 488.959,Z 169.078,A -85,B 0,C 180,E1 -6387.529,E2 -6387.529} C_VEL
LIN {X 0,Y 488.951,Z 169.081,A -85,B 0,C 180,E1 -6390.824,E2 -6390.824} C_VEL
LIN {X 0,Y 488.959,Z 169.078,A -85,B 0,C 180,E1 -6392.471,E2 -6392.471} C_VEL
LIN {X 0,Y 488.856,Z 169.089,A -85,B 0,C 180,E1 -6395.776,E2 -6395.776} C_VEL
LIN {X 0,Y 488.815,Z 169.097,A -85,B 0,C 180,E1 -6398.266,E2 -6398.266} C_VEL
LIN {X 0,Y 488.802,Z 169.095,A -85,B 0,C 180,E1 -6401.612,E2 -6401.612} C_VEL
LIN {X 0,Y 488.761,Z 169.103,A -85,B 0,C 180,E1 -6405,E2 -6405} C_VEL
LIN {X 0,Y 488.751,Z 169.108,A -85,B 0,C 180,E1 -6408.442,E2 -6408.442} C_VEL
LIN {X 0,Y 488.703,Z 169.106,A -85,B 0,C 180,E1 -6411.071,E2 -6411.071} C_VEL
LIN {X 0,Y 488.69,Z 169.109,A -85,B 0,C 180,E1 -6413.745,E2 -6413.745} C_VEL
LIN {X 0,Y 488.787,Z 169.095,A -85,B 0,C 180,E1 -6416.944,E2 -6416.944} C_VEL
LIN {X 0,Y 488.73,Z 169.109,A -85,B 0,C 180,E1 -6420.218,E2 -6420.218} C_VEL
LIN {X 0,Y 488.731,Z 169.104,A -85,B 0,C 180,E1 -6423.484,E2 -6423.484} C_VEL
LIN {X 0,Y 488.684,Z 169.11,A -85,B 0,C 180,E1 -6426.356,E2 -6426.356} C_VEL
LIN {X 0,Y 488.737,Z 169.103,A -85,B 0,C 180,E1 -6429.25,E2 -6429.25} C_VEL
LIN {X 0,Y 488.706,Z 169.111,A -85,B 0,C 180,E1 -6431.6,E2 -6431.6} C_VEL
LIN {X 0,Y 488.705,Z 169.105,A -85,B 0,C 180,E1 -6434.801,E2 -6434.801} C_VEL
LIN {X 0,Y 488.685,Z 169.115,A -85,B 0,C 180,E1 -6437.474,E2 -6437.474} C_VEL
LIN {X 0,Y 488.727,Z 169.109,A -85,B 0,C 180,E1 -6439.677,E2 -6439.677} C_VEL
LIN {X 0,Y 488.673,Z 169.109,A -85,B 0,C 180,E1 -6442.278,E2 -6442.278} C_VEL
LIN {X 0,Y 488.722,Z 169.107,A -85,B 0,C 180,E1 -6445.052,E2 -6445.052} C_VEL
LIN {X 0,Y 488.697,Z 169.106,A -85,B 0,C 180,E1 -6448.046,E2 -6448.046} C_VEL
LIN {X 0,Y 488.727,Z 169.105,A -85,B 0,C 180,E1 -6450.731,E2 -6450.731} C_VEL
LIN {X 0,Y 488.75,Z 169.102,A -85,B 0,C 180,E1 -6453.528,E2 -6453.528} C_VEL
LIN {X 0,Y 488.686,Z 169.108,A -85,B 0,C 180,E1 -6456.255,E2 -6456.255} C_VEL
LIN {X 0,Y 488.739,Z 169.106,A -85,B 0,C 180,E1 -6459.176,E2 -6459.176} C_VEL
LIN {X 0,Y 488.752,Z 169.1,A -85,B 0,C 180,E1 -6461.628,E2 -6461.628} C_VEL
LIN {X 0,Y 488.755,Z 169.104,A -85,B 0,C 180,E1 -6465,E2 -6465} C_VEL
LIN {X 0,Y 488.798,Z 169.098,A -85,B 0,C 180,E1 -6468.388,E2 -6468.388} C_VEL
LIN {X 0,Y 488.811,Z 169.092,A -85,B 0,C 180,E1 -6471.734,E2 -6471.734} C_VEL
LIN {X 0,Y 488.848,Z 169.092,A -85,B 0,C 180,E1 -6474.225,E2 -6474.225} C_VEL
LIN {X 0,Y 488.953,Z 169.074,A -85,B 0,C 180,E1 -6477.529,E2 -6477.529} C_VEL
LIN {X 0,Y 488.948,Z 169.077,A -85,B 0,C 180,E1 -6480.824,E2 -6480.824} C_VEL
LIN {X 0,Y 488.954,Z 169.079,A -85,B 0,C 180,E1 -6482.472,E2 -6482.472} C_VEL
LIN {X 0,Y 488.843,Z 169.091,A -85,B 0,C 180,E1 -6485.776,E2 -6485.776} C_VEL
LIN {X 0,Y 488.812,Z 169.097,A -85,B 0,C 180,E1 -6488.267,E2 -6488.267} C_VEL
LIN {X 0,Y 488.8,Z 169.097,A -85,B 0,C 180,E1 -6491.613,E2 -6491.613} C_VEL
LIN {X 0,Y 488.757,Z 169.099,A -85,B 0,C 180,E1 -6495.001,E2 -6495.001} C_VEL
LIN {X 0,Y 488.75,Z 169.1,A -85,B 0,C 180,E1 -6498.443,E2 -6498.443} C_VEL
LIN {X 0,Y 488.702,Z 169.107,A -85,B 0,C 180,E1 -6501.071,E2 -6501.071} C_VEL
LIN {X 0,Y 488.689,Z 169.114,A -85,B 0,C 180,E1 -6503.746,E2 -6503.746} C_VEL
LIN {X 0,Y 488.787,Z 169.097,A -85,B 0,C 180,E1 -6506.944,E2 -6506.944} C_VEL
LIN {X 0,Y 488.706,Z 169.105,A -85,B 0,C 180,E1 -6510.363,E2 -6510.363} C_VEL
LIN {X 0,Y 488.731,Z 169.109,A -85,B 0,C 180,E1 -6513.485,E2 -6513.485} C_VEL
LIN {X 0,Y 488.679,Z 169.111,A -85,B 0,C 180,E1 -6516.355,E2 -6516.355} C_VEL
LIN {X 0,Y 488.699,Z 169.114,A -85,B 0,C 180,E1 -6519.255,E2 -6519.255} C_VEL
LIN {X 0,Y 488.686,Z 169.115,A -85,B 0,C 180,E1 -6522.527,E2 -6522.527} C_VEL
LIN {X 0,Y 488.751,Z 169.503,A -85,B 0,C 180,E1 -6523.648,E2 -6523.648} C_VEL
LIN {X 0,Y 489.277,Z 172.991,A -85,B 0,C 180,E1 -6526.412,E2 -6526.412} C_VEL
LIN {X 0,Y 489.566,Z 176.072,A -85,B 0,C 180,E1 -6528.674,E2 -6528.674} C_VEL
LIN {X 0,Y 489.49,Z 179.265,A -85,B 0,C 180,E1 -6530.835,E2 -6530.835} C_VEL
LIN {X 0,Y 489.168,Z 184.144,A -85,B 0,C 180,E1 -6533.911,E2 -6533.911} C_VEL
LIN {X 0,Y 488.919,Z 189.191,A -85,B 0,C 180,E1 -6536.892,E2 -6536.892} C_VEL
LIN {X 0,Y 488.747,Z 194.344,A -85,B 0,C 180,E1 -6539.783,E2 -6539.783} C_VEL
LIN {X 0,Y 488.549,Z 200.583,A -85,B 0,C 180,E1 -6543.114,E2 -6543.114} C_VEL
LIN {X 0,Y 488.379,Z 206.704,A -85,B 0,C 180,E1 -6546.239,E2 -6546.239} C_VEL
LIN {X 0,Y 488.281,Z 213.068,A -85,B 0,C 180,E1 -6549.321,E2 -6549.321} C_VEL
LIN {X 0,Y 488.121,Z 219.461,A -85,B 0,C 180,E1 -6552.401,E2 -6552.401} C_VEL
LIN {X 0,Y 488.035,Z 225.524,A -85,B 0,C 180,E1 -6555.297,E2 -6555.297} C_VEL
LIN {X 0,Y 490.13,Z 237.258,A -85,B 0,C 180,E1 -6555.666,E2 -6555.666} C_VEL
LIN {X 0,Y 490.819,Z 242.451,A -85,B 0,C 180,E1 -6555.859,E2 -6555.859} C_VEL
LIN {X 0,Y 490.443,Z 254.366,A -85,B 0,C 180,E1 -6556.376,E2 -6556.376} C_VEL
LIN {X 0,Y 490.111,Z 264.411,A -85,B 0,C 180,E1 -6556.943,E2 -6556.943} C_VEL
LIN {X 0,Y 489.763,Z 273.461,A -85,B 0,C 180,E1 -6557.57,E2 -6557.57} C_VEL
LIN {X 0,Y 489.474,Z 282.162,A -85,B 0,C 180,E1 -6558.299,E2 -6558.299} C_VEL
LIN {X 0,Y 489.199,Z 289.531,A -85,B 0,C 180,E1 -6559.027,E2 -6559.027} C_VEL
LIN {X 0,Y 488.886,Z 296.721,A -85,B 0,C 180,E1 -6559.857,E2 -6559.857} C_VEL
LIN {X 0,Y 488.594,Z 304.267,A -85,B 0,C 180,E1 -6560.896,E2 -6560.896} C_VEL
LIN {X 0,Y 488.361,Z 310.555,A -85,B 0,C 180,E1 -6561.934,E2 -6561.934} C_VEL
LIN {X 0,Y 488.185,Z 315.789,A -85,B 0,C 180,E1 -6562.971,E2 -6562.971} C_VEL
LIN {X 0,Y 488.099,Z 320.886,A -85,B 0,C 180,E1 -6564.215,E2 -6564.215} C_VEL
LIN {X 0,Y 487.938,Z 324.843,A -85,B 0,C 180,E1 -6565.456,E2 -6565.456} C_VEL
LIN {X 0,Y 487.969,Z 327.766,A -85,B 0,C 180,E1 -6566.697,E2 -6566.697} C_VEL
LIN {X 0,Y 487.889,Z 330.193,A -85,B 0,C 180,E1 -6568.349,E2 -6568.349} C_VEL
LIN {X 0,Y 487.834,Z 330.777,A -85,B 0,C 180,E1 -6569.175,E2 -6569.175} C_VEL
LIN {X 0,Y 487.834,Z 330.777,A -85,B 0,C 180,E1 -6570.825,E2 -6570.825} C_VEL
LIN {X 0,Y 487.889,Z 330.193,A -85,B 0,C 180,E1 -6571.651,E2 -6571.651} C_VEL
LIN {X 0,Y 487.969,Z 327.766,A -85,B 0,C 180,E1 -6573.303,E2 -6573.303} C_VEL
LIN {X 0,Y 487.938,Z 324.843,A -85,B 0,C 180,E1 -6574.544,E2 -6574.544} C_VEL
LIN {X 0,Y 488.101,Z 320.886,A -85,B 0,C 180,E1 -6575.785,E2 -6575.785} C_VEL
LIN {X 0,Y 488.185,Z 315.789,A -85,B 0,C 180,E1 -6577.029,E2 -6577.029} C_VEL
LIN {X 0,Y 488.361,Z 310.555,A -85,B 0,C 180,E1 -6578.066,E2 -6578.066} C_VEL
LIN {X 0,Y 488.594,Z 304.267,A -85,B 0,C 180,E1 -6579.104,E2 -6579.104} C_VEL
LIN {X 0,Y 488.887,Z 296.721,A -85,B 0,C 180,E1 -6580.143,E2 -6580.143} C_VEL
LIN {X 0,Y 489.249,Z 287.616,A -85,B 0,C 180,E1 -6581.182,E2 -6581.182} C_VEL
LIN {X 0,Y 489.718,Z 276.158,A -85,B 0,C 180,E1 -6582.221,E2 -6582.221} C_VEL
LIN {X 0,Y 489.953,Z 267.576,A -85,B 0,C 180,E1 -6582.857,E2 -6582.857} C_VEL
LIN {X 0,Y 490.312,Z 257.382,A -85,B 0,C 180,E1 -6583.469,E2 -6583.469} C_VEL
LIN {X 0,Y 490.64,Z 247.598,A -85,B 0,C 180,E1 -6583.935,E2 -6583.935} C_VEL
LIN {X 0,Y 490.62,Z 240.295,A -85,B 0,C 180,E1 -6584.226,E2 -6584.226} C_VEL
LIN {X 0,Y 488.426,Z 227.712,A -85,B 0,C 180,E1 -6584.641,E2 -6584.641} C_VEL
LIN {X 0,Y 488.035,Z 225.524,A -85,B 0,C 180,E1 -6584.703,E2 -6584.703} C_VEL
LIN {X 0,Y 488.143,Z 218.314,A -85,B 0,C 180,E1 -6588.152,E2 -6588.152} C_VEL
LIN {X 0,Y 488.276,Z 212.215,A -85,B 0,C 180,E1 -6591.09,E2 -6591.09} C_VEL
LIN {X 0,Y 488.379,Z 206.704,A -85,B 0,C 180,E1 -6593.761,E2 -6593.761} C_VEL
LIN {X 0,Y 488.549,Z 200.583,A -85,B 0,C 180,E1 -6596.886,E2 -6596.886} C_VEL
LIN {X 0,Y 488.746,Z 194.333,A -85,B 0,C 180,E1 -6600.217,E2 -6600.217} C_VEL
LIN {X 0,Y 488.953,Z 188.46,A -85,B 0,C 180,E1 -6603.522,E2 -6603.522} C_VEL
LIN {X 0,Y 489.189,Z 183.578,A -85,B 0,C 180,E1 -6606.434,E2 -6606.434} C_VEL
LIN {X 0,Y 489.465,Z 179.239,A -85,B 0,C 180,E1 -6609.18,E2 -6609.18} C_VEL
LIN {X 0,Y 489.577,Z 175.505,A -85,B 0,C 180,E1 -6611.714,E2 -6611.714} C_VEL
LIN {X 0,Y 489.17,Z 172.327,A -85,B 0,C 180,E1 -6614.08,E2 -6614.08} C_VEL
LIN {X 0,Y 488.751,Z 169.503,A -85,B 0,C 180,E1 -6616.352,E2 -6616.352} C_VEL
LIN {X 0,Y 488.686,Z 169.113,A -85,B 0,C 180,E1 -6617.473,E2 -6617.473} C_VEL
LIN {X 0,Y 488.699,Z 169.114,A -85,B 0,C 180,E1 -6620.745,E2 -6620.745} C_VEL
LIN {X 0,Y 488.674,Z 169.11,A -85,B 0,C 180,E1 -6623.867,E2 -6623.867} C_VEL
LIN {X 0,Y 488.735,Z 169.107,A -85,B 0,C 180,E1 -6626.876,E2 -6626.876} C_VEL
LIN {X 0,Y 488.72,Z 169.104,A -85,B 0,C 180,E1 -6629.78,E2 -6629.78} C_VEL
LIN {X 0,Y 488.787,Z 169.097,A -85,B 0,C 180,E1 -6633.056,E2 -6633.056} C_VEL
LIN {X 0,Y 488.689,Z 169.114,A -85,B 0,C 180,E1 -6636.254,E2 -6636.254} C_VEL
LIN {X 0,Y 488.742,Z 169.101,A -85,B 0,C 180,E1 -6639.175,E2 -6639.175} C_VEL
LIN {X 0,Y 488.755,Z 169.1,A -85,B 0,C 180,E1 -6641.627,E2 -6641.627} C_VEL
LIN {X 0,Y 488.757,Z 169.099,A -85,B 0,C 180,E1 -6644.999,E2 -6644.999} C_VEL
LIN {X 0,Y 488.8,Z 169.097,A -85,B 0,C 180,E1 -6648.387,E2 -6648.387} C_VEL
LIN {X 0,Y 488.812,Z 169.097,A -85,B 0,C 180,E1 -6651.733,E2 -6651.733} C_VEL
LIN {X 0,Y 488.843,Z 169.091,A -85,B 0,C 180,E1 -6654.224,E2 -6654.224} C_VEL
LIN {X 0,Y 488.953,Z 169.079,A -85,B 0,C 180,E1 -6657.528,E2 -6657.528} C_VEL
LIN {X 0,Y 488.948,Z 169.075,A -85,B 0,C 180,E1 -6660.823,E2 -6660.823} C_VEL
LIN {X 0,Y 488.953,Z 169.074,A -85,B 0,C 180,E1 -6662.471,E2 -6662.471} C_VEL
LIN {X 0,Y 488.848,Z 169.092,A -85,B 0,C 180,E1 -6665.775,E2 -6665.775} C_VEL
LIN {X 0,Y 488.811,Z 169.092,A -85,B 0,C 180,E1 -6668.266,E2 -6668.266} C_VEL
LIN {X 0,Y 488.798,Z 169.098,A -85,B 0,C 180,E1 -6671.612,E2 -6671.612} C_VEL
LIN {X 0,Y 488.755,Z 169.104,A -85,B 0,C 180,E1 -6675,E2 -6675} C_VEL
LIN {X 0,Y 488.748,Z 169.101,A -85,B 0,C 180,E1 -6678.442,E2 -6678.442} C_VEL
LIN {X 0,Y 488.7,Z 169.114,A -85,B 0,C 180,E1 -6681.071,E2 -6681.071} C_VEL
LIN {X 0,Y 488.686,Z 169.108,A -85,B 0,C 180,E1 -6683.745,E2 -6683.745} C_VEL
LIN {X 0,Y 488.785,Z 169.103,A -85,B 0,C 180,E1 -6686.944,E2 -6686.944} C_VEL
LIN {X 0,Y 488.727,Z 169.104,A -85,B 0,C 180,E1 -6690.218,E2 -6690.218} C_VEL
LIN {X 0,Y 488.729,Z 169.102,A -85,B 0,C 180,E1 -6693.484,E2 -6693.484} C_VEL
LIN {X 0,Y 488.682,Z 169.113,A -85,B 0,C 180,E1 -6696.356,E2 -6696.356} C_VEL
LIN {X 0,Y 488.736,Z 169.102,A -85,B 0,C 180,E1 -6699.25,E2 -6699.25} C_VEL
LIN {X 0,Y 488.705,Z 169.105,A -85,B 0,C 180,E1 -6701.601,E2 -6701.601} C_VEL
LIN {X 0,Y 488.706,Z 169.108,A -85,B 0,C 180,E1 -6704.801,E2 -6704.801} C_VEL
LIN {X 0,Y 488.685,Z 169.108,A -85,B 0,C 180,E1 -6707.475,E2 -6707.475} C_VEL
LIN {X 0,Y 488.727,Z 169.104,A -85,B 0,C 180,E1 -6709.677,E2 -6709.677} C_VEL
LIN {X 0,Y 488.677,Z 169.109,A -85,B 0,C 180,E1 -6712.842,E2 -6712.842} C_VEL
LIN {X 0,Y 488.73,Z 169.109,A -85,B 0,C 180,E1 -6715.888,E2 -6715.888} C_VEL
LIN {X 0,Y 488.692,Z 169.107,A -85,B 0,C 180,E1 -6718.821,E2 -6718.821} C_VEL
LIN {X 0,Y 488.742,Z 169.106,A -85,B 0,C 180,E1 -6721.672,E2 -6721.672} C_VEL
LIN {X 0,Y 488.738,Z 169.102,A -85,B 0,C 180,E1 -6724.344,E2 -6724.344} C_VEL
LIN {X 0,Y 488.094,Z 169.185,A -85,B 0,C 180,E1 -6725.031,E2 -6725.031} C_VEL
LIN {X 0,Y 485.229,Z 169.548,A -85,B 0,C 180,E1 -6726.148,E2 -6726.148} C_VEL
LIN {X 0,Y 482.783,Z 169.853,A -85,B 0,C 180,E1 -6727.048,E2 -6727.048} C_VEL
LIN {X 0,Y 481.724,Z 169.982,A -85,B 0,C 180,E1 -6727.743,E2 -6727.743} C_VEL
LIN {X 0,Y 481.635,Z 169.99,A -85,B 0,C 180,E1 -6727.979,E2 -6727.979} C_VEL
LIN {X 0,Y 481.704,Z 169.978,A -85,B 0,C 180,E1 -6730.393,E2 -6730.393} C_VEL
LIN {X 0,Y 481.687,Z 169.984,A -85,B 0,C 180,E1 -6733.034,E2 -6733.034} C_VEL
LIN {X 0,Y 481.691,Z 169.986,A -85,B 0,C 180,E1 -6735.639,E2 -6735.639} C_VEL
LIN {X 0,Y 481.747,Z 169.974,A -85,B 0,C 180,E1 -6738.215,E2 -6738.215} C_VEL
LIN {X 0,Y 481.76,Z 169.976,A -85,B 0,C 180,E1 -6741.612,E2 -6741.612} C_VEL
LIN {X 0,Y 481.816,Z 169.966,A -85,B 0,C 180,E1 -6744.14,E2 -6744.14} C_VEL
LIN {X 0,Y 481.926,Z 169.955,A -85,B 0,C 180,E1 -6747.493,E2 -6747.493} C_VEL
LIN {X 0,Y 481.902,Z 169.959,A -85,B 0,C 180,E1 -6750.836,E2 -6750.836} C_VEL
LIN {X 0,Y 481.926,Z 169.955,A -85,B 0,C 180,E1 -6752.507,E2 -6752.507} C_VEL
LIN {X 0,Y 481.816,Z 169.966,A -85,B 0,C 180,E1 -6755.86,E2 -6755.86} C_VEL
LIN {X 0,Y 481.76,Z 169.976,A -85,B 0,C 180,E1 -6758.388,E2 -6758.388} C_VEL
LIN {X 0,Y 481.747,Z 169.974,A -85,B 0,C 180,E1 -6761.785,E2 -6761.785} C_VEL
LIN {X 0,Y 481.74,Z 169.976,A -85,B 0,C 180,E1 -6765.224,E2 -6765.224} C_VEL
LIN {X 0,Y 481.708,Z 169.983,A -85,B 0,C 180,E1 -6768.722,E2 -6768.722} C_VEL
LIN {X 0,Y 481.642,Z 169.985,A -85,B 0,C 180,E1 -6771.395,E2 -6771.395} C_VEL
LIN {X 0,Y 481.673,Z 169.987,A -85,B 0,C 180,E1 -6774.113,E2 -6774.113} C_VEL
LIN {X 0,Y 481.742,Z 169.972,A -85,B 0,C 180,E1 -6777.139,E2 -6777.139} C_VEL
LIN {X 0,Y 481.684,Z 169.983,A -85,B 0,C 180,E1 -6779.74,E2 -6779.74} C_VEL
LIN {X 0,Y 481.668,Z 169.983,A -85,B 0,C 180,E1 -6782.674,E2 -6782.674} C_VEL
LIN {X 0,Y 481.638,Z 169.991,A -85,B 0,C 180,E1 -6785.709,E2 -6785.709} C_VEL
LIN {X 0,Y 481.709,Z 169.979,A -85,B 0,C 180,E1 -6789.354,E2 -6789.354} C_VEL
LIN {X 0,Y 481.643,Z 169.988,A -85,B 0,C 180,E1 -6792.16,E2 -6792.16} C_VEL
LIN {X 0,Y 481.653,Z 169.991,A -85,B 0,C 180,E1 -6795.543,E2 -6795.543} C_VEL
LIN {X 0,Y 481.662,Z 169.984,A -85,B 0,C 180,E1 -6798.959,E2 -6798.959} C_VEL
LIN {X 0,Y 481.691,Z 169.983,A -85,B 0,C 180,E1 -6801.144,E2 -6801.144} C_VEL
LIN {X 0,Y 481.661,Z 169.984,A -85,B 0,C 180,E1 -6804.795,E2 -6804.795} C_VEL
LIN {X 0,Y 481.665,Z 169.99,A -85,B 0,C 180,E1 -6807.326,E2 -6807.326} C_VEL
LIN {X 0,Y 481.681,Z 169.98,A -85,B 0,C 180,E1 -6810.26,E2 -6810.26} C_VEL
LIN {X 0,Y 481.739,Z 169.981,A -85,B 0,C 180,E1 -6813.112,E2 -6813.112} C_VEL
LIN {X 0,Y 481.67,Z 169.982,A -85,B 0,C 180,E1 -6815.887,E2 -6815.887} C_VEL
LIN {X 0,Y 481.695,Z 169.985,A -85,B 0,C 180,E1 -6819.028,E2 -6819.028} C_VEL
LIN {X 0,Y 481.7,Z 169.979,A -85,B 0,C 180,E1 -6822.159,E2 -6822.159} C_VEL
LIN {X 0,Y 481.736,Z 169.982,A -85,B 0,C 180,E1 -6824.776,E2 -6824.776} C_VEL
LIN {X 0,Y 481.744,Z 169.975,A -85,B 0,C 180,E1 -6828.215,E2 -6828.215} C_VEL
LIN {X 0,Y 481.756,Z 169.971,A -85,B 0,C 180,E1 -6831.612,E2 -6831.612} C_VEL
LIN {X 0,Y 481.809,Z 169.968,A -85,B 0,C 180,E1 -6834.14,E2 -6834.14} C_VEL
LIN {X 0,Y 481.921,Z 169.95,A -85,B 0,C 180,E1 -6837.493,E2 -6837.493} C_VEL
LIN {X 0,Y 481.899,Z 169.955,A -85,B 0,C 180,E1 -6840.836,E2 -6840.836} C_VEL
LIN {X 0,Y 481.921,Z 169.955,A -85,B 0,C 180,E1 -6842.508,E2 -6842.508} C_VEL
LIN {X 0,Y 481.804,Z 169.969,A -85,B 0,C 180,E1 -6845.861,E2 -6845.861} C_VEL
LIN {X 0,Y 481.757,Z 169.975,A -85,B 0,C 180,E1 -6848.389,E2 -6848.389} C_VEL
LIN {X 0,Y 481.745,Z 169.978,A -85,B 0,C 180,E1 -6851.785,E2 -6851.785} C_VEL
LIN {X 0,Y 481.738,Z 169.974,A -85,B 0,C 180,E1 -6855.225,E2 -6855.225} C_VEL
LIN {X 0,Y 481.707,Z 169.977,A -85,B 0,C 180,E1 -6858.722,E2 -6858.722} C_VEL
LIN {X 0,Y 481.641,Z 169.989,A -85,B 0,C 180,E1 -6861.395,E2 -6861.395} C_VEL
LIN {X 0,Y 481.673,Z 169.983,A -85,B 0,C 180,E1 -6864.114,E2 -6864.114} C_VEL
LIN {X 0,Y 481.741,Z 169.976,A -85,B 0,C 180,E1 -6867.139,E2 -6867.139} C_VEL
LIN {X 0,Y 481.674,Z 169.985,A -85,B 0,C 180,E1 -6869.742,E2 -6869.742} C_VEL
LIN {X 0,Y 481.668,Z 169.983,A -85,B 0,C 180,E1 -6872.675,E2 -6872.675} C_VEL
LIN {X 0,Y 481.633,Z 169.991,A -85,B 0,C 180,E1 -6875.71,E2 -6875.71} C_VEL
LIN {X 0,Y 481.669,Z 169.989,A -85,B 0,C 180,E1 -6878.86,E2 -6878.86} C_VEL
LIN {X 0,Y 481.644,Z 169.991,A -85,B 0,C 180,E1 -6881.913,E2 -6881.913} C_VEL
LIN {X 0,Y 481.707,Z 170.338,A -85,B 0,C 180,E1 -6883.293,E2 -6883.293} C_VEL
LIN {X 0,Y 482.369,Z 174.661,A -85,B 0,C 180,E1 -6886.783,E2 -6886.783} C_VEL
LIN {X 0,Y 482.553,Z 178.045,A -85,B 0,C 180,E1 -6889.231,E2 -6889.231} C_VEL
LIN {X 0,Y 482.378,Z 181.989,A -85,B 0,C 180,E1 -6891.884,E2 -6891.884} C_VEL
LIN {X 0,Y 482.01,Z 187.554,A -85,B 0,C 180,E1 -6895.345,E2 -6895.345} C_VEL
LIN {X 0,Y 481.766,Z 192.628,A -85,B 0,C 180,E1 -6898.321,E2 -6898.321} C_VEL
LIN {X 0,Y 481.578,Z 197.836,A -85,B 0,C 180,E1 -6901.211,E2 -6901.211} C_VEL
LIN {X 0,Y 481.43,Z 203.1,A -85,B 0,C 180,E1 -6904.028,E2 -6904.028} C_VEL
LIN {X 0,Y 481.28,Z 208.724,A -85,B 0,C 180,E1 -6906.923,E2 -6906.923} C_VEL
LIN {X 0,Y 481.186,Z 213.942,A -85,B 0,C 180,E1 -6909.48,E2 -6909.48} C_VEL
LIN {X 0,Y 481.045,Z 219.433,A -85,B 0,C 180,E1 -6912.133,E2 -6912.133} C_VEL
LIN {X 0,Y 480.995,Z 225.524,A -85,B 0,C 180,E1 -6915.077,E2 -6915.077} C_VEL
LIN {X 0,Y 483.063,Z 237.107,A -85,B 0,C 180,E1 -6915.448,E2 -6915.448} C_VEL
LIN {X 0,Y 483.87,Z 243.73,A -85,B 0,C 180,E1 -6915.705,E2 -6915.705} C_VEL
LIN {X 0,Y 483.554,Z 254.357,A -85,B 0,C 180,E1 -6916.178,E2 -6916.178} C_VEL
LIN {X 0,Y 483.163,Z 264.804,A -85,B 0,C 180,E1 -6916.778,E2 -6916.778} C_VEL
LIN {X 0,Y 482.792,Z 273.453,A -85,B 0,C 180,E1 -6917.388,E2 -6917.388} C_VEL
LIN {X 0,Y 482.507,Z 282.156,A -85,B 0,C 180,E1 -6918.127,E2 -6918.127} C_VEL
LIN {X 0,Y 482.19,Z 289.526,A -85,B 0,C 180,E1 -6918.865,E2 -6918.865} C_VEL
LIN {X 0,Y 481.872,Z 296.717,A -85,B 0,C 180,E1 -6919.708,E2 -6919.708} C_VEL
LIN {X 0,Y 481.577,Z 304.263,A -85,B 0,C 180,E1 -6920.762,E2 -6920.762} C_VEL
LIN {X 0,Y 481.325,Z 310.551,A -85,B 0,C 180,E1 -6921.816,E2 -6921.816} C_VEL
LIN {X 0,Y 481.101,Z 315.784,A -85,B 0,C 180,E1 -6922.867,E2 -6922.867} C_VEL
LIN {X 0,Y 480.989,Z 319.532,A -85,B 0,C 180,E1 -6923.761,E2 -6923.761} C_VEL
LIN {X 0,Y 480.906,Z 323.631,A -85,B 0,C 180,E1 -6924.97,E2 -6924.97} C_VEL
LIN {X 0,Y 480.855,Z 325.975,A -85,B 0,C 180,E1 -6925.809,E2 -6925.809} C_VEL
LIN {X 0,Y 480.894,Z 327.763,A -85,B 0,C 180,E1 -6926.649,E2 -6926.649} C_VEL
LIN {X 0,Y 480.79,Z 330.19,A -85,B 0,C 180,E1 -6928.325,E2 -6928.325} C_VEL
LIN {X 0,Y 480.76,Z 330.773,A -85,B 0,C 180,E1 -6929.162,E2 -6929.162} C_VEL
LIN {X 0,Y 480.76,Z 330.773,A -85,B 0,C 180,E1 -6930.838,E2 -6930.838} C_VEL
LIN {X 0,Y 480.79,Z 330.19,A -85,B 0,C 180,E1 -6931.675,E2 -6931.675} C_VEL
LIN {X 0,Y 480.894,Z 327.763,A -85,B 0,C 180,E1 -6933.351,E2 -6933.351} C_VEL
LIN {X 0,Y 480.853,Z 324.84,A -85,B 0,C 180,E1 -6934.611,E2 -6934.611} C_VEL
LIN {X 0,Y 481.019,Z 320.882,A -85,B 0,C 180,E1 -6935.87,E2 -6935.87} C_VEL
LIN {X 0,Y 481.061,Z 317.685,A -85,B 0,C 180,E1 -6936.712,E2 -6936.712} C_VEL
LIN {X 0,Y 481.249,Z 311.701,A -85,B 0,C 180,E1 -6937.975,E2 -6937.975} C_VEL
LIN {X 0,Y 481.524,Z 305.633,A -85,B 0,C 180,E1 -6939.027,E2 -6939.027} C_VEL
LIN {X 0,Y 481.828,Z 298.338,A -85,B 0,C 180,E1 -6940.08,E2 -6940.08} C_VEL
LIN {X 0,Y 482.099,Z 291.439,A -85,B 0,C 180,E1 -6940.924,E2 -6940.924} C_VEL
LIN {X 0,Y 482.453,Z 283.287,A -85,B 0,C 180,E1 -6941.767,E2 -6941.767} C_VEL
LIN {X 0,Y 482.786,Z 274.802,A -85,B 0,C 180,E1 -6942.506,E2 -6942.506} C_VEL
LIN {X 0,Y 483.061,Z 266.596,A -85,B 0,C 180,E1 -6943.107,E2 -6943.107} C_VEL
LIN {X 0,Y 483.421,Z 256.368,A -85,B 0,C 180,E1 -6943.718,E2 -6943.718} C_VEL
LIN {X 0,Y 483.741,Z 247.588,A -85,B 0,C 180,E1 -6944.138,E2 -6944.138} C_VEL
LIN {X 0,Y 483.892,Z 242.444,A -85,B 0,C 180,E1 -6944.348,E2 -6944.348} C_VEL
LIN {X 0,Y 481.55,Z 228.687,A -85,B 0,C 180,E1 -6944.834,E2 -6944.834} C_VEL
LIN {X 0,Y 480.995,Z 225.524,A -85,B 0,C 180,E1 -6944.923,E2 -6944.923} C_VEL
LIN {X 0,Y 481.064,Z 218.601,A -85,B 0,C 180,E1 -6948.267,E2 -6948.267} C_VEL
LIN {X 0,Y 481.214,Z 212.108,A -85,B 0,C 180,E1 -6951.415,E2 -6951.415} C_VEL
LIN {X 0,Y 481.342,Z 206.608,A -85,B 0,C 180,E1 -6954.131,E2 -6954.131} C_VEL
LIN {X 0,Y 481.507,Z 200.995,A -85,B 0,C 180,E1 -6957.083,E2 -6957.083} C_VEL
LIN {X 0,Y 481.624,Z 196.044,A -85,B 0,C 180,E1 -6959.744,E2 -6959.744} C_VEL
LIN {X 0,Y 481.845,Z 190.907,A -85,B 0,C 180,E1 -6962.66,E2 -6962.66} C_VEL
LIN {X 0,Y 482.097,Z 185.843,A -85,B 0,C 180,E1 -6965.67,E2 -6965.67} C_VEL
LIN {X 0,Y 482.423,Z 180.954,A -85,B 0,C 180,E1 -6968.786,E2 -6968.786} C_VEL
LIN {X 0,Y 482.556,Z 177.753,A -85,B 0,C 180,E1 -6970.948,E2 -6970.948} C_VEL
LIN {X 0,Y 482.363,Z 174.626,A -85,B 0,C 180,E1 -6973.239,E2 -6973.239} C_VEL
LIN {X 0,Y 481.911,Z 171.647,A -85,B 0,C 180,E1 -6975.609,E2 -6975.609} C_VEL
LIN {X 0,Y 481.667,Z 170.165,A -85,B 0,C 180,E1 -6976.848,E2 -6976.848} C_VEL
LIN {X 0,Y 481.666,Z 169.987,A -85,B 0,C 180,E1 -6980.058,E2 -6980.058} C_VEL
LIN {X 0,Y 481.623,Z 169.99,A -85,B 0,C 180,E1 -6983.252,E2 -6983.252} C_VEL
LIN {X 0,Y 481.707,Z 169.98,A -85,B 0,C 180,E1 -6986.329,E2 -6986.329} C_VEL
LIN {X 0,Y 481.647,Z 169.985,A -85,B 0,C 180,E1 -6989.417,E2 -6989.417} C_VEL
LIN {X 0,Y 481.694,Z 169.982,A -85,B 0,C 180,E1 -6992.167,E2 -6992.167} C_VEL
LIN {X 0,Y 481.714,Z 169.978,A -85,B 0,C 180,E1 -6994.969,E2 -6994.969} C_VEL
LIN {X 0,Y 481.646,Z 169.986,A -85,B 0,C 180,E1 -6997.704,E2 -6997.704} C_VEL
LIN {X 0,Y 481.7,Z 169.984,A -85,B 0,C 180,E1 -7000.392,E2 -7000.392} C_VEL
LIN {X 0,Y 481.683,Z 169.98,A -85,B 0,C 180,E1 -7003.033,E2 -7003.033} C_VEL
LIN {X 0,Y 481.684,Z 169.982,A -85,B 0,C 180,E1 -7005.638,E2 -7005.638} C_VEL
LIN {X 0,Y 481.745,Z 169.978,A -85,B 0,C 180,E1 -7008.215,E2 -7008.215} C_VEL
LIN {X 0,Y 481.757,Z 169.975,A -85,B 0,C 180,E1 -7011.611,E2 -7011.611} C_VEL
LIN {X 0,Y 481.804,Z 169.969,A -85,B 0,C 180,E1 -7014.139,E2 -7014.139} C_VEL
LIN {X 0,Y 481.92,Z 169.955,A -85,B 0,C 180,E1 -7017.492,E2 -7017.492} C_VEL
LIN {X 0,Y 481.899,Z 169.953,A -85,B 0,C 180,E1 -7020.835,E2 -7020.835} C_VEL
LIN {X 0,Y 481.921,Z 169.95,A -85,B 0,C 180,E1 -7022.507,E2 -7022.507} C_VEL
LIN {X 0,Y 481.809,Z 169.968,A -85,B 0,C 180,E1 -7025.86,E2 -7025.86} C_VEL
LIN {X 0,Y 481.756,Z 169.971,A -85,B 0,C 180,E1 -7028.388,E2 -7028.388} C_VEL
LIN {X 0,Y 481.744,Z 169.975,A -85,B 0,C 180,E1 -7031.785,E2 -7031.785} C_VEL
LIN {X 0,Y 481.736,Z 169.982,A -85,B 0,C 180,E1 -7035.224,E2 -7035.224} C_VEL
LIN {X 0,Y 481.706,Z 169.98,A -85,B 0,C 180,E1 -7038.721,E2 -7038.721} C_VEL
LIN {X 0,Y 481.639,Z 169.989,A -85,B 0,C 180,E1 -7041.394,E2 -7041.394} C_VEL
LIN {X 0,Y 481.67,Z 169.982,A -85,B 0,C 180,E1 -7044.113,E2 -7044.113} C_VEL
LIN {X 0,Y 481.74,Z 169.977,A -85,B 0,C 180,E1 -7047.139,E2 -7047.139} C_VEL
LIN {X 0,Y 481.681,Z 169.98,A -85,B 0,C 180,E1 -7049.74,E2 -7049.74} C_VEL
LIN {X 0,Y 481.665,Z 169.99,A -85,B 0,C 180,E1 -7052.674,E2 -7052.674} C_VEL
LIN {X 0,Y 481.636,Z 169.986,A -85,B 0,C 180,E1 -7055.709,E2 -7055.709} C_VEL
LIN {X 0,Y 481.708,Z 169.977,A -85,B 0,C 180,E1 -7059.354,E2 -7059.354} C_VEL
LIN {X 0,Y 481.642,Z 169.99,A -85,B 0,C 180,E1 -7062.161,E2 -7062.161} C_VEL
LIN {X 0,Y 481.653,Z 169.984,A -85,B 0,C 180,E1 -7065.543,E2 -7065.543} C_VEL
LIN {X 0,Y 481.651,Z 169.984,A -85,B 0,C 180,E1 -7068.958,E2 -7068.958} C_VEL
LIN {X 0,Y 481.651,Z 169.99,A -85,B 0,C 180,E1 -7071.993,E2 -7071.993} C_VEL
LIN {X 0,Y 481.688,Z 169.98,A -85,B 0,C 180,E1 -7075.318,E2 -7075.318} C_VEL
LIN {X 0,Y 481.644,Z 169.988,A -85,B 0,C 180,E1 -7078.312,E2 -7078.312} C_VEL
LIN {X 0,Y 481.702,Z 169.979,A -85,B 0,C 180,E1 -7081.219,E2 -7081.219} C_VEL
LIN {X 0,Y 481.696,Z 169.983,A -85,B 0,C 180,E1 -7084.043,E2 -7084.043} C_VEL
LIN {X 0,Y 481.67,Z 169.982,A -85,B 0,C 180,E1 -7086.812,E2 -7086.812} C_VEL
LIN {X 0,Y 481.635,Z 169.99,A -85,B 0,C 180,E1 -7087.979,E2 -7087.979} C_VEL
LIN {X 0,Y 480.965,Z 170.07,A -85,B 0,C 180,E1 -7088.677,E2 -7088.677} C_VEL
LIN {X 0,Y 478.137,Z 170.428,A -85,B 0,C 180,E1 -7089.811,E2 -7089.811} C_VEL
LIN {X 0,Y 475.753,Z 170.725,A -85,B 0,C 180,E1 -7090.725,E2 -7090.725} C_VEL
LIN {X 0,Y 474.733,Z 170.852,A -85,B 0,C 180,E1 -7091.431,E2 -7091.431} C_VEL
LIN {X 0,Y 474.651,Z 170.861,A -85,B 0,C 180,E1 -7091.67,E2 -7091.67} C_VEL
LIN {X 0,Y 474.697,Z 170.853,A -85,B 0,C 180,E1 -7094.544,E2 -7094.544} C_VEL
LIN {X 0,Y 474.701,Z 170.853,A -85,B 0,C 180,E1 -7098.038,E2 -7098.038} C_VEL
LIN {X 0,Y 474.725,Z 170.853,A -85,B 0,C 180,E1 -7101.487,E2 -7101.487} C_VEL
LIN {X 0,Y 474.778,Z 170.843,A -85,B 0,C 180,E1 -7104.052,E2 -7104.052} C_VEL
LIN {X 0,Y 474.892,Z 170.832,A -85,B 0,C 180,E1 -7107.455,E2 -7107.455} C_VEL
LIN {X 0,Y 474.909,Z 170.828,A -85,B 0,C 180,E1 -7110,E2 -7110} C_VEL
LIN {X 0,Y 474.892,Z 170.832,A -85,B 0,C 180,E1 -7112.545,E2 -7112.545} C_VEL
LIN {X 0,Y 474.778,Z 170.843,A -85,B 0,C 180,E1 -7115.948,E2 -7115.948} C_VEL
LIN {X 0,Y 474.725,Z 170.853,A -85,B 0,C 180,E1 -7118.513,E2 -7118.513} C_VEL
LIN {X 0,Y 474.701,Z 170.853,A -85,B 0,C 180,E1 -7121.962,E2 -7121.962} C_VEL
LIN {X 0,Y 474.697,Z 170.853,A -85,B 0,C 180,E1 -7125.456,E2 -7125.456} C_VEL
LIN {X 0,Y 474.661,Z 170.857,A -85,B 0,C 180,E1 -7129.01,E2 -7129.01} C_VEL
LIN {X 0,Y 474.586,Z 170.865,A -85,B 0,C 180,E1 -7131.729,E2 -7131.729} C_VEL
LIN {X 0,Y 474.655,Z 170.861,A -85,B 0,C 180,E1 -7134.493,E2 -7134.493} C_VEL
LIN {X 0,Y 474.694,Z 170.851,A -85,B 0,C 180,E1 -7137.339,E2 -7137.339} C_VEL
LIN {X 0,Y 474.605,Z 170.862,A -85,B 0,C 180,E1 -7140.811,E2 -7140.811} C_VEL
LIN {X 0,Y 474.634,Z 170.866,A -85,B 0,C 180,E1 -7143.984,E2 -7143.984} C_VEL
LIN {X 0,Y 474.57,Z 170.866,A -85,B 0,C 180,E1 -7146.9,E2 -7146.9} C_VEL
LIN {X 0,Y 474.645,Z 170.863,A -85,B 0,C 180,E1 -7149.651,E2 -7149.651} C_VEL
LIN {X 0,Y 474.609,Z 170.862,A -85,B 0,C 180,E1 -7152.934,E2 -7152.934} C_VEL
LIN {X 0,Y 474.603,Z 170.866,A -85,B 0,C 180,E1 -7155.895,E2 -7155.895} C_VEL
LIN {X 0,Y 474.634,Z 170.86,A -85,B 0,C 180,E1 -7159.039,E2 -7159.039} C_VEL
LIN {X 0,Y 474.61,Z 170.866,A -85,B 0,C 180,E1 -7161.703,E2 -7161.703} C_VEL
LIN {X 0,Y 474.623,Z 170.86,A -85,B 0,C 180,E1 -7164.726,E2 -7164.726} C_VEL
LIN {X 0,Y 474.629,Z 170.861,A -85,B 0,C 180,E1 -7167.788,E2 -7167.788} C_VEL
LIN {X 0,Y 474.626,Z 170.863,A -85,B 0,C 180,E1 -7170.883,E2 -7170.883} C_VEL
LIN {X 0,Y 474.653,Z 170.857,A -85,B 0,C 180,E1 -7173.629,E2 -7173.629} C_VEL
LIN {X 0,Y 474.629,Z 170.862,A -85,B 0,C 180,E1 -7176.641,E2 -7176.641} C_VEL
LIN {X 0,Y 474.65,Z 170.856,A -85,B 0,C 180,E1 -7180.09,E2 -7180.09} C_VEL
LIN {X 0,Y 474.644,Z 170.864,A -85,B 0,C 180,E1 -7182.775,E2 -7182.775} C_VEL
LIN {X 0,Y 474.641,Z 170.858,A -85,B 0,C 180,E1 -7185.421,E2 -7185.421} C_VEL
LIN {X 0,Y 474.697,Z 170.851,A -85,B 0,C 180,E1 -7188.038,E2 -7188.038} C_VEL
LIN {X 0,Y 474.722,Z 170.847,A -85,B 0,C 180,E1 -7191.487,E2 -7191.487} C_VEL
LIN {X 0,Y 474.772,Z 170.843,A -85,B 0,C 180,E1 -7194.053,E2 -7194.053} C_VEL
LIN {X 0,Y 474.887,Z 170.827,A -85,B 0,C 180,E1 -7197.456,E2 -7197.456} C_VEL
LIN {X 0,Y 474.904,Z 170.828,A -85,B 0,C 180,E1 -7200,E2 -7200} C_VEL
LIN {X 0,Y 474.887,Z 170.831,A -85,B 0,C 180,E1 -7202.545,E2 -7202.545} C_VEL
LIN {X 0,Y 474.766,Z 170.847,A -85,B 0,C 180,E1 -7205.948,E2 -7205.948} C_VEL
LIN {X 0,Y 474.722,Z 170.85,A -85,B 0,C 180,E1 -7208.514,E2 -7208.514} C_VEL
LIN {X 0,Y 474.699,Z 170.858,A -85,B 0,C 180,E1 -7211.963,E2 -7211.963} C_VEL
LIN {X 0,Y 474.695,Z 170.853,A -85,B 0,C 180,E1 -7215.456,E2 -7215.456} C_VEL
LIN {X 0,Y 474.66,Z 170.855,A -85,B 0,C 180,E1 -7219.011,E2 -7219.011} C_VEL
LIN {X 0,Y 474.585,Z 170.872,A -85,B 0,C 180,E1 -7221.73,E2 -7221.73} C_VEL
LIN {X 0,Y 474.655,Z 170.855,A -85,B 0,C 180,E1 -7224.494,E2 -7224.494} C_VEL
LIN {X 0,Y 474.676,Z 170.859,A -85,B 0,C 180,E1 -7227.335,E2 -7227.335} C_VEL
LIN {X 0,Y 474.6,Z 170.864,A -85,B 0,C 180,E1 -7230.811,E2 -7230.811} C_VEL
LIN {X 0,Y 474.634,Z 170.861,A -85,B 0,C 180,E1 -7233.984,E2 -7233.984} C_VEL
LIN {X 0,Y 474.569,Z 170.873,A -85,B 0,C 180,E1 -7236.9,E2 -7236.9} C_VEL
LIN {X 0,Y 474.611,Z 170.868,A -85,B 0,C 180,E1 -7239.646,E2 -7239.646} C_VEL
LIN {X 0,Y 474.6,Z 170.869,A -85,B 0,C 180,E1 -7242.234,E2 -7242.234} C_VEL
LIN {X 0,Y 474.63,Z 171.158,A -85,B 0,C 180,E1 -7242.933,E2 -7242.933} C_VEL
LIN {X 0,Y 475.199,Z 174.809,A -85,B 0,C 180,E1 -7245.965,E2 -7245.965} C_VEL
LIN {X 0,Y 475.527,Z 177.899,A -85,B 0,C 180,E1 -7248.313,E2 -7248.313} C_VEL
LIN {X 0,Y 475.467,Z 181.059,A -85,B 0,C 180,E1 -7250.537,E2 -7250.537} C_VEL
LIN {X 0,Y 475.197,Z 184.806,A -85,B 0,C 180,E1 -7253.001,E2 -7253.001} C_VEL
LIN {X 0,Y 474.93,Z 189.555,A -85,B 0,C 180,E1 -7255.965,E2 -7255.965} C_VEL
LIN {X 0,Y 474.665,Z 195.035,A -85,B 0,C 180,E1 -7259.178,E2 -7259.178} C_VEL
LIN {X 0,Y 474.46,Z 201.39,A -85,B 0,C 180,E1 -7262.718,E2 -7262.718} C_VEL
LIN {X 0,Y 474.278,Z 206.604,A -85,B 0,C 180,E1 -7265.487,E2 -7265.487} C_VEL
LIN {X 0,Y 474.151,Z 212.001,A -85,B 0,C 180,E1 -7268.25,E2 -7268.25} C_VEL
LIN {X 0,Y 474.018,Z 217.499,A -85,B 0,C 180,E1 -7270.963,E2 -7270.963} C_VEL
LIN {X 0,Y 473.942,Z 225.398,A -85,B 0,C 180,E1 -7274.805,E2 -7274.805} C_VEL
LIN {X 0,Y 473.941,Z 225.53,A -85,B 0,C 180,E1 -7274.859,E2 -7274.859} C_VEL
LIN {X 0,Y 475.811,Z 235.679,A -85,B 0,C 180,E1 -7275.177,E2 -7275.177} C_VEL
LIN {X 0,Y 476.987,Z 243.72,A -85,B 0,C 180,E1 -7275.494,E2 -7275.494} C_VEL
LIN {X 0,Y 476.657,Z 254.348,A -85,B 0,C 180,E1 -7275.974,E2 -7275.974} C_VEL
LIN {X 0,Y 476.263,Z 264.473,A -85,B 0,C 180,E1 -7276.561,E2 -7276.561} C_VEL
LIN {X 0,Y 475.852,Z 273.446,A -85,B 0,C 180,E1 -7277.201,E2 -7277.201} C_VEL
LIN {X 0,Y 475.542,Z 282.199,A -85,B 0,C 180,E1 -7277.956,E2 -7277.956} C_VEL
LIN {X 0,Y 475.215,Z 289.52,A -85,B 0,C 180,E1 -7278.7,E2 -7278.7} C_VEL
LIN {X 0,Y 474.86,Z 296.713,A -85,B 0,C 180,E1 -7279.555,E2 -7279.555} C_VEL
LIN {X 0,Y 474.605,Z 302.889,A -85,B 0,C 180,E1 -7280.41,E2 -7280.41} C_VEL
LIN {X 0,Y 474.316,Z 309.396,A -85,B 0,C 180,E1 -7281.479,E2 -7281.479} C_VEL
LIN {X 0,Y 474.102,Z 313.875,A -85,B 0,C 180,E1 -7282.333,E2 -7282.333} C_VEL
LIN {X 0,Y 473.958,Z 318.792,A -85,B 0,C 180,E1 -7283.465,E2 -7283.465} C_VEL
LIN {X 0,Y 473.845,Z 323.628,A -85,B 0,C 180,E1 -7284.895,E2 -7284.895} C_VEL
LIN {X 0,Y 473.759,Z 325.974,A -85,B 0,C 180,E1 -7285.746,E2 -7285.746} C_VEL
LIN {X 0,Y 473.802,Z 327.76,A -85,B 0,C 180,E1 -7286.599,E2 -7286.599} C_VEL
LIN {X 0,Y 473.695,Z 330.186,A -85,B 0,C 180,E1 -7288.3,E2 -7288.3} C_VEL
LIN {X 0,Y 473.688,Z 330.769,A -85,B 0,C 180,E1 -7289.15,E2 -7289.15} C_VEL
LIN {X 0,Y 473.688,Z 330.769,A -85,B 0,C 180,E1 -7290.85,E2 -7290.85} C_VEL
LIN {X 0,Y 473.695,Z 330.186,A -85,B 0,C 180,E1 -7291.7,E2 -7291.7} C_VEL
LIN {X 0,Y 473.802,Z 327.76,A -85,B 0,C 180,E1 -7293.401,E2 -7293.401} C_VEL
LIN {X 0,Y 473.775,Z 324.836,A -85,B 0,C 180,E1 -7294.68,E2 -7294.68} C_VEL
LIN {X 0,Y 473.939,Z 320.877,A -85,B 0,C 180,E1 -7295.958,E2 -7295.958} C_VEL
LIN {X 0,Y 474.03,Z 315.78,A -85,B 0,C 180,E1 -7297.24,E2 -7297.24} C_VEL
LIN {X 0,Y 474.266,Z 310.546,A -85,B 0,C 180,E1 -7298.307,E2 -7298.307} C_VEL
LIN {X 0,Y 474.55,Z 304.259,A -85,B 0,C 180,E1 -7299.376,E2 -7299.376} C_VEL
LIN {X 0,Y 474.795,Z 298.333,A -85,B 0,C 180,E1 -7300.231,E2 -7300.231} C_VEL
LIN {X 0,Y 475.105,Z 291.433,A -85,B 0,C 180,E1 -7301.087,E2 -7301.087} C_VEL
LIN {X 0,Y 475.489,Z 283.281,A -85,B 0,C 180,E1 -7301.942,E2 -7301.942} C_VEL
LIN {X 0,Y 475.85,Z 274.552,A -85,B 0,C 180,E1 -7302.71,E2 -7302.71} C_VEL
LIN {X 0,Y 476.151,Z 266.587,A -85,B 0,C 180,E1 -7303.301,E2 -7303.301} C_VEL
LIN {X 0,Y 476.537,Z 256.359,A -85,B 0,C 180,E1 -7303.92,E2 -7303.92} C_VEL
LIN {X 0,Y 476.926,Z 246.292,A -85,B 0,C 180,E1 -7304.399,E2 -7304.399} C_VEL
LIN {X 0,Y 476.657,Z 241.123,A -85,B 0,C 180,E1 -7304.623,E2 -7304.623} C_VEL
LIN {X 0,Y 474.37,Z 228.093,A -85,B 0,C 180,E1 -7305.075,E2 -7305.075} C_VEL
LIN {X 0,Y 473.92,Z 225.453,A -85,B 0,C 180,E1 -7305.169,E2 -7305.169} C_VEL
LIN {X 0,Y 473.996,Z 218.825,A -85,B 0,C 180,E1 -7308.388,E2 -7308.388} C_VEL
LIN {X 0,Y 474.145,Z 213.588,A -85,B 0,C 180,E1 -7310.961,E2 -7310.961} C_VEL
LIN {X 0,Y 474.21,Z 208.358,A -85,B 0,C 180,E1 -7313.587,E2 -7313.587} C_VEL
LIN {X 0,Y 474.391,Z 203.051,A -85,B 0,C 180,E1 -7316.387,E2 -7316.387} C_VEL
LIN {X 0,Y 474.535,Z 197.781,A -85,B 0,C 180,E1 -7319.257,E2 -7319.257} C_VEL
LIN {X 0,Y 474.808,Z 192.176,A -85,B 0,C 180,E1 -7322.466,E2 -7322.466} C_VEL
LIN {X 0,Y 475.07,Z 187.067,A -85,B 0,C 180,E1 -7325.546,E2 -7325.546} C_VEL
LIN {X 0,Y 475.371,Z 182.616,A -85,B 0,C 180,E1 -7328.411,E2 -7328.411} C_VEL
LIN {X 0,Y 475.55,Z 178.708,A -85,B 0,C 180,E1 -7331.087,E2 -7331.087} C_VEL
LIN {X 0,Y 475.291,Z 175.4,A -85,B 0,C 180,E1 -7333.568,E2 -7333.568} C_VEL
LIN {X 0,Y 474.724,Z 171.833,A -85,B 0,C 180,E1 -7336.502,E2 -7336.502} C_VEL
LIN {X 0,Y 474.63,Z 171.17,A -85,B 0,C 180,E1 -7337.067,E2 -7337.067} C_VEL
LIN {X 0,Y 474.62,Z 170.867,A -85,B 0,C 180,E1 -7339.041,E2 -7339.041} C_VEL
LIN {X 0,Y 474.607,Z 170.865,A -85,B 0,C 180,E1 -7341.703,E2 -7341.703} C_VEL
LIN {X 0,Y 474.621,Z 170.868,A -85,B 0,C 180,E1 -7344.725,E2 -7344.725} C_VEL
LIN {X 0,Y 474.632,Z 170.858,A -85,B 0,C 180,E1 -7347.787,E2 -7347.787} C_VEL
LIN {X 0,Y 474.618,Z 170.864,A -85,B 0,C 180,E1 -7350.884,E2 -7350.884} C_VEL
LIN {X 0,Y 474.656,Z 170.855,A -85,B 0,C 180,E1 -7353.628,E2 -7353.628} C_VEL
LIN {X 0,Y 474.632,Z 170.863,A -85,B 0,C 180,E1 -7356.641,E2 -7356.641} C_VEL
LIN {X 0,Y 474.65,Z 170.862,A -85,B 0,C 180,E1 -7360.089,E2 -7360.089} C_VEL
LIN {X 0,Y 474.643,Z 170.858,A -85,B 0,C 180,E1 -7362.774,E2 -7362.774} C_VEL
LIN {X 0,Y 474.642,Z 170.858,A -85,B 0,C 180,E1 -7365.42,E2 -7365.42} C_VEL
LIN {X 0,Y 474.699,Z 170.858,A -85,B 0,C 180,E1 -7368.037,E2 -7368.037} C_VEL
LIN {X 0,Y 474.722,Z 170.85,A -85,B 0,C 180,E1 -7371.486,E2 -7371.486} C_VEL
LIN {X 0,Y 474.766,Z 170.847,A -85,B 0,C 180,E1 -7374.052,E2 -7374.052} C_VEL
LIN {X 0,Y 474.887,Z 170.831,A -85,B 0,C 180,E1 -7377.455,E2 -7377.455} C_VEL
LIN {X 0,Y 474.904,Z 170.828,A -85,B 0,C 180,E1 -7380,E2 -7380} C_VEL
LIN {X 0,Y 474.887,Z 170.827,A -85,B 0,C 180,E1 -7382.544,E2 -7382.544} C_VEL
LIN {X 0,Y 474.772,Z 170.843,A -85,B 0,C 180,E1 -7385.947,E2 -7385.947} C_VEL
LIN {X 0,Y 474.722,Z 170.847,A -85,B 0,C 180,E1 -7388.513,E2 -7388.513} C_VEL
LIN {X 0,Y 474.697,Z 170.851,A -85,B 0,C 180,E1 -7391.962,E2 -7391.962} C_VEL
LIN {X 0,Y 474.693,Z 170.856,A -85,B 0,C 180,E1 -7395.455,E2 -7395.455} C_VEL
LIN {X 0,Y 474.659,Z 170.862,A -85,B 0,C 180,E1 -7399.01,E2 -7399.01} C_VEL
LIN {X 0,Y 474.582,Z 170.865,A -85,B 0,C 180,E1 -7401.729,E2 -7401.729} C_VEL
LIN {X 0,Y 474.652,Z 170.858,A -85,B 0,C 180,E1 -7404.493,E2 -7404.493} C_VEL
LIN {X 0,Y 474.692,Z 170.853,A -85,B 0,C 180,E1 -7407.339,E2 -7407.339} C_VEL
LIN {X 0,Y 474.603,Z 170.87,A -85,B 0,C 180,E1 -7410.811,E2 -7410.811} C_VEL
LIN {X 0,Y 474.631,Z 170.859,A -85,B 0,C 180,E1 -7413.984,E2 -7413.984} C_VEL
LIN {X 0,Y 474.569,Z 170.87,A -85,B 0,C 180,E1 -7416.9,E2 -7416.9} C_VEL
LIN {X 0,Y 474.644,Z 170.857,A -85,B 0,C 180,E1 -7419.651,E2 -7419.651} C_VEL
LIN {X 0,Y 474.608,Z 170.863,A -85,B 0,C 180,E1 -7422.934,E2 -7422.934} C_VEL
LIN {X 0,Y 474.603,Z 170.865,A -85,B 0,C 180,E1 -7425.895,E2 -7425.895} C_VEL
LIN {X 0,Y 474.622,Z 170.86,A -85,B 0,C 180,E1 -7429.041,E2 -7429.041} C_VEL
LIN {X 0,Y 474.605,Z 170.864,A -85,B 0,C 180,E1 -7431.704,E2 -7431.704} C_VEL
LIN {X 0,Y 474.625,Z 170.86,A -85,B 0,C 180,E1 -7434.726,E2 -7434.726} C_VEL
LIN {X 0,Y 474.633,Z 170.864,A -85,B 0,C 180,E1 -7437.788,E2 -7437.788} C_VEL
LIN {X 0,Y 474.627,Z 170.859,A -85,B 0,C 180,E1 -7440.883,E2 -7440.883} C_VEL
LIN {X 0,Y 474.657,Z 170.861,A -85,B 0,C 180,E1 -7443.629,E2 -7443.629} C_VEL
LIN {X 0,Y 474.631,Z 170.858,A -85,B 0,C 180,E1 -7446.641,E2 -7446.641} C_VEL
LIN {X 0,Y 474.652,Z 170.86,A -85,B 0,C 180,E1 -7450.09,E2 -7450.09} C_VEL
LIN {X 0,Y 474.651,Z 170.861,A -85,B 0,C 180,E1 -7451.67,E2 -7451.67} C_VEL
LIN {X 0,Y 473.989,Z 170.946,A -85,B 0,C 180,E1 -7452.379,E2 -7452.379} C_VEL
LIN {X 0,Y 471.14,Z 171.304,A -85,B 0,C 180,E1 -7453.53,E2 -7453.53} C_VEL
LIN {X 0,Y 468.725,Z 171.604,A -85,B 0,C 180,E1 -7454.459,E2 -7454.459} C_VEL
LIN {X 0,Y 467.683,Z 171.731,A -85,B 0,C 180,E1 -7455.176,E2 -7455.176} C_VEL
LIN {X 0,Y 467.596,Z 171.74,A -85,B 0,C 180,E1 -7455.419,E2 -7455.419} C_VEL
LIN {X 0,Y 467.65,Z 171.732,A -85,B 0,C 180,E1 -7458.734,E2 -7458.734} C_VEL
LIN {X 0,Y 467.745,Z 171.72,A -85,B 0,C 180,E1 -7462.228,E2 -7462.228} C_VEL
LIN {X 0,Y 467.723,Z 171.725,A -85,B 0,C 180,E1 -7464.828,E2 -7464.828} C_VEL
LIN {X 0,Y 467.857,Z 171.709,A -85,B 0,C 180,E1 -7467.417,E2 -7467.417} C_VEL
LIN {X 0,Y 467.88,Z 171.704,A -85,B 0,C 180,E1 -7470,E2 -7470} C_VEL
LIN {X 0,Y 467.857,Z 171.709,A -85,B 0,C 180,E1 -7472.583,E2 -7472.583} C_VEL
LIN {X 0,Y 467.743,Z 171.72,A -85,B 0,C 180,E1 -7476.037,E2 -7476.037} C_VEL
LIN {X 0,Y 467.678,Z 171.732,A -85,B 0,C 180,E1 -7478.643,E2 -7478.643} C_VEL
LIN {X 0,Y 467.652,Z 171.732,A -85,B 0,C 180,E1 -7482.145,E2 -7482.145} C_VEL
LIN {X 0,Y 467.636,Z 171.733,A -85,B 0,C 180,E1 -7485.695,E2 -7485.695} C_VEL
LIN {X 0,Y 467.614,Z 171.739,A -85,B 0,C 180,E1 -7488.765,E2 -7488.765} C_VEL
LIN {X 0,Y 467.577,Z 171.737,A -85,B 0,C 180,E1 -7491.268,E2 -7491.268} C_VEL
LIN {X 0,Y 467.569,Z 171.742,A -85,B 0,C 180,E1 -7493.943,E2 -7493.943} C_VEL
LIN {X 0,Y 467.612,Z 171.734,A -85,B 0,C 180,E1 -7496.8,E2 -7496.8} C_VEL
LIN {X 0,Y 467.583,Z 171.74,A -85,B 0,C 180,E1 -7499.736,E2 -7499.736} C_VEL
LIN {X 0,Y 467.579,Z 171.737,A -85,B 0,C 180,E1 -7502.758,E2 -7502.758} C_VEL
LIN {X 0,Y 467.551,Z 171.748,A -85,B 0,C 180,E1 -7505.889,E2 -7505.889} C_VEL
LIN {X 0,Y 467.594,Z 171.736,A -85,B 0,C 180,E1 -7509.143,E2 -7509.143} C_VEL
LIN {X 0,Y 467.58,Z 171.737,A -85,B 0,C 180,E1 -7512.567,E2 -7512.567} C_VEL
LIN {X 0,Y 467.564,Z 171.74,A -85,B 0,C 180,E1 -7515.053,E2 -7515.053} C_VEL
LIN {X 0,Y 467.582,Z 171.743,A -85,B 0,C 180,E1 -7517.44,E2 -7517.44} C_VEL
LIN {X 0,Y 467.609,Z 171.734,A -85,B 0,C 180,E1 -7520.859,E2 -7520.859} C_VEL
LIN {X 0,Y 467.556,Z 171.74,A -85,B 0,C 180,E1 -7524.26,E2 -7524.26} C_VEL
LIN {X 0,Y 467.575,Z 171.745,A -85,B 0,C 180,E1 -7527.321,E2 -7527.321} C_VEL
LIN {X 0,Y 467.571,Z 171.74,A -85,B 0,C 180,E1 -7530.666,E2 -7530.666} C_VEL
LIN {X 0,Y 467.61,Z 171.74,A -85,B 0,C 180,E1 -7533.2,E2 -7533.2} C_VEL
LIN {X 0,Y 467.586,Z 171.738,A -85,B 0,C 180,E1 -7536.468,E2 -7536.468} C_VEL
LIN {X 0,Y 467.617,Z 171.732,A -85,B 0,C 180,E1 -7539.777,E2 -7539.777} C_VEL
LIN {X 0,Y 467.602,Z 171.738,A -85,B 0,C 180,E1 -7542.507,E2 -7542.507} C_VEL
LIN {X 0,Y 467.599,Z 171.737,A -85,B 0,C 180,E1 -7545.197,E2 -7545.197} C_VEL
LIN {X 0,Y 467.649,Z 171.728,A -85,B 0,C 180,E1 -7547.855,E2 -7547.855} C_VEL
LIN {X 0,Y 467.675,Z 171.725,A -85,B 0,C 180,E1 -7551.358,E2 -7551.358} C_VEL
LIN {X 0,Y 467.736,Z 171.719,A -85,B 0,C 180,E1 -7553.963,E2 -7553.963} C_VEL
LIN {X 0,Y 467.853,Z 171.703,A -85,B 0,C 180,E1 -7557.418,E2 -7557.418} C_VEL
LIN {X 0,Y 467.875,Z 171.704,A -85,B 0,C 180,E1 -7560,E2 -7560} C_VEL
LIN {X 0,Y 467.852,Z 171.706,A -85,B 0,C 180,E1 -7562.583,E2 -7562.583} C_VEL
LIN {X 0,Y 467.731,Z 171.725,A -85,B 0,C 180,E1 -7566.038,E2 -7566.038} C_VEL
LIN {X 0,Y 467.676,Z 171.726,A -85,B 0,C 180,E1 -7568.643,E2 -7568.643} C_VEL
LIN {X 0,Y 467.651,Z 171.733,A -85,B 0,C 180,E1 -7572.146,E2 -7572.146} C_VEL
LIN {X 0,Y 467.634,Z 171.736,A -85,B 0,C 180,E1 -7575.696,E2 -7575.696} C_VEL
LIN {X 0,Y 467.612,Z 171.733,A -85,B 0,C 180,E1 -7578.765,E2 -7578.765} C_VEL
LIN {X 0,Y 467.576,Z 171.74,A -85,B 0,C 180,E1 -7581.269,E2 -7581.269} C_VEL
LIN {X 0,Y 467.569,Z 171.742,A -85,B 0,C 180,E1 -7583.944,E2 -7583.944} C_VEL
LIN {X 0,Y 467.612,Z 171.733,A -85,B 0,C 180,E1 -7586.801,E2 -7586.801} C_VEL
LIN {X 0,Y 467.549,Z 171.744,A -85,B 0,C 180,E1 -7589.739,E2 -7589.739} C_VEL
LIN {X 0,Y 467.58,Z 171.738,A -85,B 0,C 180,E1 -7592.759,E2 -7592.759} C_VEL
LIN {X 0,Y 467.551,Z 171.745,A -85,B 0,C 180,E1 -7595.89,E2 -7595.89} C_VEL
LIN {X 0,Y 467.571,Z 171.746,A -85,B 0,C 180,E1 -7599.146,E2 -7599.146} C_VEL
LIN {X 0,Y 467.571,Z 171.745,A -85,B 0,C 180,E1 -7601.404,E2 -7601.404} C_VEL
LIN {X 0,Y 467.585,Z 171.995,A -85,B 0,C 180,E1 -7602.568,E2 -7602.568} C_VEL
LIN {X 0,Y 468.054,Z 174.958,A -85,B 0,C 180,E1 -7605.113,E2 -7605.113} C_VEL
LIN {X 0,Y 468.464,Z 178.005,A -85,B 0,C 180,E1 -7607.539,E2 -7607.539} C_VEL
LIN {X 0,Y 468.505,Z 181.278,A -85,B 0,C 180,E1 -7609.912,E2 -7609.912} C_VEL
LIN {X 0,Y 468.209,Z 185.386,A -85,B 0,C 180,E1 -7612.708,E2 -7612.708} C_VEL
LIN {X 0,Y 467.909,Z 190.11,A -85,B 0,C 180,E1 -7615.701,E2 -7615.701} C_VEL
LIN {X 0,Y 467.65,Z 195.484,A -85,B 0,C 180,E1 -7618.939,E2 -7618.939} C_VEL
LIN {X 0,Y 467.412,Z 201.247,A -85,B 0,C 180,E1 -7622.218,E2 -7622.218} C_VEL
LIN {X 0,Y 467.239,Z 206.531,A -85,B 0,C 180,E1 -7625.092,E2 -7625.092} C_VEL
LIN {X 0,Y 467.068,Z 211.894,A -85,B 0,C 180,E1 -7627.903,E2 -7627.903} C_VEL
LIN {X 0,Y 466.94,Z 217.394,A -85,B 0,C 180,E1 -7630.663,E2 -7630.663} C_VEL
LIN {X 0,Y 466.806,Z 222.856,A -85,B 0,C 180,E1 -7633.378,E2 -7633.378} C_VEL
LIN {X 0,Y 466.83,Z 225.449,A -85,B 0,C 180,E1 -7634.625,E2 -7634.625} C_VEL
LIN {X 0,Y 468.686,Z 235.356,A -85,B 0,C 180,E1 -7634.943,E2 -7634.943} C_VEL
LIN {X 0,Y 470.069,Z 244.851,A -85,B 0,C 180,E1 -7635.331,E2 -7635.331} C_VEL
LIN {X 0,Y 469.726,Z 255.218,A -85,B 0,C 180,E1 -7635.818,E2 -7635.818} C_VEL
LIN {X 0,Y 469.348,Z 264.359,A -85,B 0,C 180,E1 -7636.359,E2 -7636.359} C_VEL
LIN {X 0,Y 468.915,Z 273.355,A -85,B 0,C 180,E1 -7637.008,E2 -7637.008} C_VEL
LIN {X 0,Y 468.591,Z 282.225,A -85,B 0,C 180,E1 -7637.782,E2 -7637.782} C_VEL
LIN {X 0,Y 468.249,Z 289.491,A -85,B 0,C 180,E1 -7638.529,E2 -7638.529} C_VEL
LIN {X 0,Y 467.839,Z 296.708,A -85,B 0,C 180,E1 -7639.396,E2 -7639.396} C_VEL
LIN {X 0,Y 467.582,Z 302.885,A -85,B 0,C 180,E1 -7640.265,E2 -7640.265} C_VEL
LIN {X 0,Y 467.287,Z 309.392,A -85,B 0,C 180,E1 -7641.35,E2 -7641.35} C_VEL
LIN {X 0,Y 467.046,Z 313.87,A -85,B 0,C 180,E1 -7642.217,E2 -7642.217} C_VEL
LIN {X 0,Y 466.867,Z 319.206,A -85,B 0,C 180,E1 -7643.483,E2 -7643.483} C_VEL
LIN {X 0,Y 466.783,Z 323.624,A -85,B 0,C 180,E1 -7644.817,E2 -7644.817} C_VEL
LIN {X 0,Y 466.668,Z 325.972,A -85,B 0,C 180,E1 -7645.682,E2 -7645.682} C_VEL
LIN {X 0,Y 466.698,Z 327.757,A -85,B 0,C 180,E1 -7646.547,E2 -7646.547} C_VEL
LIN {X 0,Y 466.604,Z 330.182,A -85,B 0,C 180,E1 -7648.274,E2 -7648.274} C_VEL
LIN {X 0,Y 466.59,Z 330.765,A -85,B 0,C 180,E1 -7649.137,E2 -7649.137} C_VEL
LIN {X 0,Y 466.59,Z 330.765,A -85,B 0,C 180,E1 -7650.863,E2 -7650.863} C_VEL
LIN {X 0,Y 466.604,Z 330.182,A -85,B 0,C 180,E1 -7651.726,E2 -7651.726} C_VEL
LIN {X 0,Y 466.698,Z 327.757,A -85,B 0,C 180,E1 -7653.453,E2 -7653.453} C_VEL
LIN {X 0,Y 466.703,Z 324.832,A -85,B 0,C 180,E1 -7654.751,E2 -7654.751} C_VEL
LIN {X 0,Y 466.836,Z 320.873,A -85,B 0,C 180,E1 -7656.049,E2 -7656.049} C_VEL
LIN {X 0,Y 466.96,Z 315.775,A -85,B 0,C 180,E1 -7657.35,E2 -7657.35} C_VEL
LIN {X 0,Y 467.207,Z 310.542,A -85,B 0,C 180,E1 -7658.434,E2 -7658.434} C_VEL
LIN {X 0,Y 467.507,Z 304.255,A -85,B 0,C 180,E1 -7659.518,E2 -7659.518} C_VEL
LIN {X 0,Y 467.771,Z 298.329,A -85,B 0,C 180,E1 -7660.387,E2 -7660.387} C_VEL
LIN {X 0,Y 468.12,Z 291.41,A -85,B 0,C 180,E1 -7661.255,E2 -7661.255} C_VEL
LIN {X 0,Y 468.525,Z 283.226,A -85,B 0,C 180,E1 -7662.122,E2 -7662.122} C_VEL
LIN {X 0,Y 468.869,Z 274.465,A -85,B 0,C 180,E1 -7662.903,E2 -7662.903} C_VEL
LIN {X 0,Y 469.251,Z 265.992,A -85,B 0,C 180,E1 -7663.533,E2 -7663.533} C_VEL
LIN {X 0,Y 469.657,Z 256.224,A -85,B 0,C 180,E1 -7664.129,E2 -7664.129} C_VEL
LIN {X 0,Y 470.033,Z 246.139,A -85,B 0,C 180,E1 -7664.614,E2 -7664.614} C_VEL
LIN {X 0,Y 469.251,Z 238.76,A -85,B 0,C 180,E1 -7664.931,E2 -7664.931} C_VEL
LIN {X 0,Y 467.13,Z 227.207,A -85,B 0,C 180,E1 -7665.328,E2 -7665.328} C_VEL
LIN {X 0,Y 466.834,Z 225.312,A -85,B 0,C 180,E1 -7665.404,E2 -7665.404} C_VEL
LIN {X 0,Y 466.916,Z 219.059,A -85,B 0,C 180,E1 -7668.508,E2 -7668.508} C_VEL
LIN {X 0,Y 467.077,Z 213.73,A -85,B 0,C 180,E1 -7671.169,E2 -7671.169} C_VEL
LIN {X 0,Y 467.164,Z 208.306,A -85,B 0,C 180,E1 -7673.965,E2 -7673.965} C_VEL
LIN {X 0,Y 467.346,Z 202.989,A -85,B 0,C 180,E1 -7676.817,E2 -7676.817} C_VEL
LIN {X 0,Y 467.52,Z 197.759,A -85,B 0,C 180,E1 -7679.74,E2 -7679.74} C_VEL
LIN {X 0,Y 467.78,Z 192.635,A -85,B 0,C 180,E1 -7682.742,E2 -7682.742} C_VEL
LIN {X 0,Y 468.066,Z 187.61,A -85,B 0,C 180,E1 -7685.844,E2 -7685.844} C_VEL
LIN {X 0,Y 468.401,Z 182.728,A -85,B 0,C 180,E1 -7689.063,E2 -7689.063} C_VEL
LIN {X 0,Y 468.548,Z 179.406,A -85,B 0,C 180,E1 -7691.411,E2 -7691.411} C_VEL
LIN {X 0,Y 468.244,Z 176.165,A -85,B 0,C 180,E1 -7693.908,E2 -7693.908} C_VEL
LIN {X 0,Y 467.769,Z 173.319,A -85,B 0,C 180,E1 -7696.28,E2 -7696.28} C_VEL
LIN {X 0,Y 467.587,Z 171.988,A -85,B 0,C 180,E1 -7697.439,E2 -7697.439} C_VEL
LIN {X 0,Y 467.571,Z 171.743,A -85,B 0,C 180,E1 -7700.046,E2 -7700.046} C_VEL
LIN {X 0,Y 467.527,Z 171.749,A -85,B 0,C 180,E1 -7703.037,E2 -7703.037} C_VEL
LIN {X 0,Y 467.583,Z 171.739,A -85,B 0,C 180,E1 -7706.211,E2 -7706.211} C_VEL
LIN {X 0,Y 467.566,Z 171.739,A -85,B 0,C 180,E1 -7709.265,E2 -7709.265} C_VEL
LIN {X 0,Y 467.629,Z 171.738,A -85,B 0,C 180,E1 -7712.461,E2 -7712.461} C_VEL
LIN {X 0,Y 467.599,Z 171.735,A -85,B 0,C 180,E1 -7715.112,E2 -7715.112} C_VEL
LIN {X 0,Y 467.531,Z 171.746,A -85,B 0,C 180,E1 -7717.926,E2 -7717.926} C_VEL
LIN {X 0,Y 467.619,Z 171.735,A -85,B 0,C 180,E1 -7720.692,E2 -7720.692} C_VEL
LIN {X 0,Y 467.645,Z 171.736,A -85,B 0,C 180,E1 -7724.114,E2 -7724.114} C_VEL
LIN {X 0,Y 467.649,Z 171.731,A -85,B 0,C 180,E1 -7727.642,E2 -7727.642} C_VEL
LIN {X 0,Y 467.659,Z 171.729,A -85,B 0,C 180,E1 -7730.484,E2 -7730.484} C_VEL
LIN {X 0,Y 467.696,Z 171.723,A -85,B 0,C 180,E1 -7733.095,E2 -7733.095} C_VEL
LIN {X 0,Y 467.716,Z 171.72,A -85,B 0,C 180,E1 -7734.827,E2 -7734.827} C_VEL
LIN {X 0,Y 467.852,Z 171.706,A -85,B 0,C 180,E1 -7737.417,E2 -7737.417} C_VEL
LIN {X 0,Y 467.875,Z 171.704,A -85,B 0,C 180,E1 -7740,E2 -7740} C_VEL
LIN {X 0,Y 467.853,Z 171.703,A -85,B 0,C 180,E1 -7742.582,E2 -7742.582} C_VEL
LIN {X 0,Y 467.736,Z 171.719,A -85,B 0,C 180,E1 -7746.037,E2 -7746.037} C_VEL
LIN {X 0,Y 467.675,Z 171.725,A -85,B 0,C 180,E1 -7748.642,E2 -7748.642} C_VEL
LIN {X 0,Y 467.649,Z 171.728,A -85,B 0,C 180,E1 -7752.145,E2 -7752.145} C_VEL
LIN {X 0,Y 467.632,Z 171.732,A -85,B 0,C 180,E1 -7755.695,E2 -7755.695} C_VEL
LIN {X 0,Y 467.611,Z 171.736,A -85,B 0,C 180,E1 -7758.764,E2 -7758.764} C_VEL
LIN {X 0,Y 467.574,Z 171.743,A -85,B 0,C 180,E1 -7761.268,E2 -7761.268} C_VEL
LIN {X 0,Y 467.566,Z 171.738,A -85,B 0,C 180,E1 -7763.943,E2 -7763.943} C_VEL
LIN {X 0,Y 467.61,Z 171.74,A -85,B 0,C 180,E1 -7766.8,E2 -7766.8} C_VEL
LIN {X 0,Y 467.58,Z 171.737,A -85,B 0,C 180,E1 -7769.736,E2 -7769.736} C_VEL
LIN {X 0,Y 467.576,Z 171.745,A -85,B 0,C 180,E1 -7772.758,E2 -7772.758} C_VEL
LIN {X 0,Y 467.55,Z 171.741,A -85,B 0,C 180,E1 -7775.889,E2 -7775.889} C_VEL
LIN {X 0,Y 467.609,Z 171.734,A -85,B 0,C 180,E1 -7779.141,E2 -7779.141} C_VEL
LIN {X 0,Y 467.58,Z 171.743,A -85,B 0,C 180,E1 -7782.567,E2 -7782.567} C_VEL
LIN {X 0,Y 467.564,Z 171.739,A -85,B 0,C 180,E1 -7785.053,E2 -7785.053} C_VEL
LIN {X 0,Y 467.583,Z 171.737,A -85,B 0,C 180,E1 -7787.44,E2 -7787.44} C_VEL
LIN {X 0,Y 467.577,Z 171.738,A -85,B 0,C 180,E1 -7790.855,E2 -7790.855} C_VEL
LIN {X 0,Y 467.558,Z 171.745,A -85,B 0,C 180,E1 -7794.26,E2 -7794.26} C_VEL
LIN {X 0,Y 467.577,Z 171.738,A -85,B 0,C 180,E1 -7797.321,E2 -7797.321} C_VEL
LIN {X 0,Y 467.573,Z 171.738,A -85,B 0,C 180,E1 -7800.666,E2 -7800.666} C_VEL
LIN {X 0,Y 467.612,Z 171.734,A -85,B 0,C 180,E1 -7803.2,E2 -7803.2} C_VEL
LIN {X 0,Y 467.589,Z 171.736,A -85,B 0,C 180,E1 -7806.468,E2 -7806.468} C_VEL
LIN {X 0,Y 467.62,Z 171.739,A -85,B 0,C 180,E1 -7809.777,E2 -7809.777} C_VEL
LIN {X 0,Y 467.605,Z 171.737,A -85,B 0,C 180,E1 -7812.507,E2 -7812.507} C_VEL
LIN {X 0,Y 467.596,Z 171.74,A -85,B 0,C 180,E1 -7815.419,E2 -7815.419} C_VEL
LIN {X 0,Y 466.925,Z 171.823,A -85,B 0,C 180,E1 -7816.138,E2 -7816.138} C_VEL
LIN {X 0,Y 464.081,Z 172.18,A -85,B 0,C 180,E1 -7817.306,E2 -7817.306} C_VEL
LIN {X 0,Y 461.682,Z 172.476,A -85,B 0,C 180,E1 -7818.248,E2 -7818.248} C_VEL
LIN {X 0,Y 460.656,Z 172.605,A -85,B 0,C 180,E1 -7818.976,E2 -7818.976} C_VEL
LIN {X 0,Y 460.574,Z 172.614,A -85,B 0,C 180,E1 -7819.222,E2 -7819.222} C_VEL
LIN {X 0,Y 460.716,Z 172.596,A -85,B 0,C 180,E1 -7822.538,E2 -7822.538} C_VEL
LIN {X 0,Y 460.696,Z 172.599,A -85,B 0,C 180,E1 -7824.748,E2 -7824.748} C_VEL
LIN {X 0,Y 460.822,Z 172.586,A -85,B 0,C 180,E1 -7827.378,E2 -7827.378} C_VEL
LIN {X 0,Y 460.85,Z 172.579,A -85,B 0,C 180,E1 -7830,E2 -7830} C_VEL
LIN {X 0,Y 460.822,Z 172.585,A -85,B 0,C 180,E1 -7832.622,E2 -7832.622} C_VEL
LIN {X 0,Y 460.708,Z 172.597,A -85,B 0,C 180,E1 -7836.13,E2 -7836.13} C_VEL
LIN {X 0,Y 460.625,Z 172.611,A -85,B 0,C 180,E1 -7838.776,E2 -7838.776} C_VEL
LIN {X 0,Y 460.609,Z 172.611,A -85,B 0,C 180,E1 -7842.445,E2 -7842.445} C_VEL
LIN {X 0,Y 460.596,Z 172.612,A -85,B 0,C 180,E1 -7845.997,E2 -7845.997} C_VEL
LIN {X 0,Y 460.567,Z 172.615,A -85,B 0,C 180,E1 -7848.902,E2 -7848.902} C_VEL
LIN {X 0,Y 460.512,Z 172.617,A -85,B 0,C 180,E1 -7851.485,E2 -7851.485} C_VEL
LIN {X 0,Y 460.538,Z 172.621,A -85,B 0,C 180,E1 -7854.332,E2 -7854.332} C_VEL
LIN {X 0,Y 460.575,Z 172.609,A -85,B 0,C 180,E1 -7857.243,E2 -7857.243} C_VEL
LIN {X 0,Y 460.523,Z 172.622,A -85,B 0,C 180,E1 -7860.239,E2 -7860.239} C_VEL
LIN {X 0,Y 460.524,Z 172.617,A -85,B 0,C 180,E1 -7863.325,E2 -7863.325} C_VEL
LIN {X 0,Y 460.474,Z 172.623,A -85,B 0,C 180,E1 -7866.529,E2 -7866.529} C_VEL
LIN {X 0,Y 460.569,Z 172.618,A -85,B 0,C 180,E1 -7869.858,E2 -7869.858} C_VEL
LIN {X 0,Y 460.507,Z 172.618,A -85,B 0,C 180,E1 -7872.9,E2 -7872.9} C_VEL
LIN {X 0,Y 460.505,Z 172.623,A -85,B 0,C 180,E1 -7875.83,E2 -7875.83} C_VEL
LIN {X 0,Y 460.533,Z 172.616,A -85,B 0,C 180,E1 -7878.99,E2 -7878.99} C_VEL
LIN {X 0,Y 460.537,Z 172.619,A -85,B 0,C 180,E1 -7881.269,E2 -7881.269} C_VEL
LIN {X 0,Y 460.507,Z 172.618,A -85,B 0,C 180,E1 -7884.555,E2 -7884.555} C_VEL
LIN {X 0,Y 460.525,Z 172.618,A -85,B 0,C 180,E1 -7887.716,E2 -7887.716} C_VEL
LIN {X 0,Y 460.541,Z 172.616,A -85,B 0,C 180,E1 -7890.77,E2 -7890.77} C_VEL
LIN {X 0,Y 460.556,Z 172.613,A -85,B 0,C 180,E1 -7893.735,E2 -7893.735} C_VEL
LIN {X 0,Y 460.539,Z 172.617,A -85,B 0,C 180,E1 -7896.624,E2 -7896.624} C_VEL
LIN {X 0,Y 460.545,Z 172.615,A -85,B 0,C 180,E1 -7899.453,E2 -7899.453} C_VEL
LIN {X 0,Y 460.552,Z 172.613,A -85,B 0,C 180,E1 -7902.23,E2 -7902.23} C_VEL
LIN {X 0,Y 460.558,Z 172.617,A -85,B 0,C 180,E1 -7904.965,E2 -7904.965} C_VEL
LIN {X 0,Y 460.604,Z 172.612,A -85,B 0,C 180,E1 -7908.56,E2 -7908.56} C_VEL
LIN {X 0,Y 460.689,Z 172.598,A -85,B 0,C 180,E1 -7912.109,E2 -7912.109} C_VEL
LIN {X 0,Y 460.69,Z 172.599,A -85,B 0,C 180,E1 -7914.749,E2 -7914.749} C_VEL
LIN {X 0,Y 460.794,Z 172.582,A -85,B 0,C 180,E1 -7917.378,E2 -7917.378} C_VEL
LIN {X 0,Y 460.846,Z 172.579,A -85,B 0,C 180,E1 -7920,E2 -7920} C_VEL
LIN {X 0,Y 460.793,Z 172.585,A -85,B 0,C 180,E1 -7922.623,E2 -7922.623} C_VEL
LIN {X 0,Y 460.697,Z 172.602,A -85,B 0,C 180,E1 -7926.131,E2 -7926.131} C_VEL
LIN {X 0,Y 460.623,Z 172.604,A -85,B 0,C 180,E1 -7928.777,E2 -7928.777} C_VEL
LIN {X 0,Y 460.608,Z 172.607,A -85,B 0,C 180,E1 -7932.445,E2 -7932.445} C_VEL
LIN {X 0,Y 460.596,Z 172.613,A -85,B 0,C 180,E1 -7935.998,E2 -7935.998} C_VEL
LIN {X 0,Y 460.566,Z 172.611,A -85,B 0,C 180,E1 -7938.902,E2 -7938.902} C_VEL
LIN {X 0,Y 460.512,Z 172.623,A -85,B 0,C 180,E1 -7941.486,E2 -7941.486} C_VEL
LIN {X 0,Y 460.538,Z 172.614,A -85,B 0,C 180,E1 -7944.333,E2 -7944.333} C_VEL
LIN {X 0,Y 460.568,Z 172.615,A -85,B 0,C 180,E1 -7947.245,E2 -7947.245} C_VEL
LIN {X 0,Y 460.507,Z 172.618,A -85,B 0,C 180,E1 -7950.241,E2 -7950.241} C_VEL
LIN {X 0,Y 460.526,Z 172.624,A -85,B 0,C 180,E1 -7953.326,E2 -7953.326} C_VEL
LIN {X 0,Y 460.474,Z 172.626,A -85,B 0,C 180,E1 -7956.53,E2 -7956.53} C_VEL
LIN {X 0,Y 460.522,Z 172.623,A -85,B 0,C 180,E1 -7959.864,E2 -7959.864} C_VEL
LIN {X 0,Y 460.52,Z 172.812,A -85,B 0,C 180,E1 -7962.182,E2 -7962.182} C_VEL
LIN {X 0,Y 461.129,Z 176.626,A -85,B 0,C 180,E1 -7965.487,E2 -7965.487} C_VEL
LIN {X 0,Y 461.474,Z 179.667,A -85,B 0,C 180,E1 -7967.926,E2 -7967.926} C_VEL
LIN {X 0,Y 461.446,Z 182.821,A -85,B 0,C 180,E1 -7970.233,E2 -7970.233} C_VEL
LIN {X 0,Y 461.215,Z 186.048,A -85,B 0,C 180,E1 -7972.446,E2 -7972.446} C_VEL
LIN {X 0,Y 460.883,Z 190.987,A -85,B 0,C 180,E1 -7975.653,E2 -7975.653} C_VEL
LIN {X 0,Y 460.608,Z 196.054,A -85,B 0,C 180,E1 -7978.75,E2 -7978.75} C_VEL
LIN {X 0,Y 460.376,Z 201.202,A -85,B 0,C 180,E1 -7981.756,E2 -7981.756} C_VEL
LIN {X 0,Y 460.215,Z 206.454,A -85,B 0,C 180,E1 -7984.686,E2 -7984.686} C_VEL
LIN {X 0,Y 460.017,Z 211.777,A -85,B 0,C 180,E1 -7987.546,E2 -7987.546} C_VEL
LIN {X 0,Y 459.887,Z 217.184,A -85,B 0,C 180,E1 -7990.355,E2 -7990.355} C_VEL
LIN {X 0,Y 459.725,Z 222.64,A -85,B 0,C 180,E1 -7993.115,E2 -7993.115} C_VEL
LIN {X 0,Y 459.738,Z 225.28,A -85,B 0,C 180,E1 -7994.383,E2 -7994.383} C_VEL
LIN {X 0,Y 461.734,Z 235.917,A -85,B 0,C 180,E1 -7994.736,E2 -7994.736} C_VEL
LIN {X 0,Y 463.088,Z 244.636,A -85,B 0,C 180,E1 -7995.105,E2 -7995.105} C_VEL
LIN {X 0,Y 462.871,Z 253.999,A -85,B 0,C 180,E1 -7995.548,E2 -7995.548} C_VEL
LIN {X 0,Y 462.427,Z 264.143,A -85,B 0,C 180,E1 -7996.151,E2 -7996.151} C_VEL
LIN {X 0,Y 461.983,Z 273.144,A -85,B 0,C 180,E1 -7996.81,E2 -7996.81} C_VEL
LIN {X 0,Y 461.654,Z 281.169,A -85,B 0,C 180,E1 -7997.513,E2 -7997.513} C_VEL
LIN {X 0,Y 461.256,Z 289.278,A -85,B 0,C 180,E1 -7998.353,E2 -7998.353} C_VEL
LIN {X 0,Y 460.849,Z 296.5,A -85,B 0,C 180,E1 -7999.233,E2 -7999.233} C_VEL
LIN {X 0,Y 460.554,Z 302.706,A -85,B 0,C 180,E1 -8000.115,E2 -8000.115} C_VEL
LIN {X 0,Y 460.235,Z 309.246,A -85,B 0,C 180,E1 -8001.216,E2 -8001.216} C_VEL
LIN {X 0,Y 459.983,Z 313.748,A -85,B 0,C 180,E1 -8002.096,E2 -8002.096} C_VEL
LIN {X 0,Y 459.783,Z 319.515,A -85,B 0,C 180,E1 -8003.495,E2 -8003.495} C_VEL
LIN {X 0,Y 459.699,Z 323.566,A -85,B 0,C 180,E1 -8004.737,E2 -8004.737} C_VEL
LIN {X 0,Y 459.584,Z 325.929,A -85,B 0,C 180,E1 -8005.615,E2 -8005.615} C_VEL
LIN {X 0,Y 459.594,Z 327.728,A -85,B 0,C 180,E1 -8006.493,E2 -8006.493} C_VEL
LIN {X 0,Y 459.517,Z 330.169,A -85,B 0,C 180,E1 -8008.247,E2 -8008.247} C_VEL
LIN {X 0,Y 459.495,Z 330.755,A -85,B 0,C 180,E1 -8009.124,E2 -8009.124} C_VEL
LIN {X 0,Y 459.495,Z 330.755,A -85,B 0,C 180,E1 -8010.876,E2 -8010.876} C_VEL
LIN {X 0,Y 459.517,Z 330.169,A -85,B 0,C 180,E1 -8011.753,E2 -8011.753} C_VEL
LIN {X 0,Y 459.594,Z 327.728,A -85,B 0,C 180,E1 -8013.507,E2 -8013.507} C_VEL
LIN {X 0,Y 459.634,Z 324.781,A -85,B 0,C 180,E1 -8014.824,E2 -8014.824} C_VEL
LIN {X 0,Y 459.754,Z 320.795,A -85,B 0,C 180,E1 -8016.143,E2 -8016.143} C_VEL
LIN {X 0,Y 459.884,Z 315.663,A -85,B 0,C 180,E1 -8017.464,E2 -8017.464} C_VEL
LIN {X 0,Y 460.174,Z 310.402,A -85,B 0,C 180,E1 -8018.563,E2 -8018.563} C_VEL
LIN {X 0,Y 460.478,Z 304.083,A -85,B 0,C 180,E1 -8019.665,E2 -8019.665} C_VEL
LIN {X 0,Y 460.737,Z 298.127,A -85,B 0,C 180,E1 -8020.547,E2 -8020.547} C_VEL
LIN {X 0,Y 461.117,Z 291.197,A -85,B 0,C 180,E1 -8021.428,E2 -8021.428} C_VEL
LIN {X 0,Y 461.557,Z 283.014,A -85,B 0,C 180,E1 -8022.308,E2 -8022.308} C_VEL
LIN {X 0,Y 461.91,Z 274.577,A -85,B 0,C 180,E1 -8023.074,E2 -8023.074} C_VEL
LIN {X 0,Y 462.335,Z 265.775,A -85,B 0,C 180,E1 -8023.74,E2 -8023.74} C_VEL
LIN {X 0,Y 462.735,Z 256.012,A -85,B 0,C 180,E1 -8024.344,E2 -8024.344} C_VEL
LIN {X 0,Y 463.108,Z 247.216,A -85,B 0,C 180,E1 -8024.782,E2 -8024.782} C_VEL
LIN {X 0,Y 462.719,Z 242.043,A -85,B 0,C 180,E1 -8025.02,E2 -8025.02} C_VEL
LIN {X 0,Y 460.289,Z 228.332,A -85,B 0,C 180,E1 -8025.533,E2 -8025.533} C_VEL
LIN {X 0,Y 459.732,Z 225.134,A -85,B 0,C 180,E1 -8025.63,E2 -8025.63} C_VEL
LIN {X 0,Y 459.847,Z 219.007,A -85,B 0,C 180,E1 -8028.72,E2 -8028.72} C_VEL
LIN {X 0,Y 460.002,Z 213.564,A -85,B 0,C 180,E1 -8031.51,E2 -8031.51} C_VEL
LIN {X 0,Y 460.134,Z 208.212,A -85,B 0,C 180,E1 -8034.355,E2 -8034.355} C_VEL
LIN {X 0,Y 460.349,Z 202.171,A -85,B 0,C 180,E1 -8037.69,E2 -8037.69} C_VEL
LIN {X 0,Y 460.519,Z 197.743,A -85,B 0,C 180,E1 -8040.239,E2 -8040.239} C_VEL
LIN {X 0,Y 460.759,Z 192.638,A -85,B 0,C 180,E1 -8043.305,E2 -8043.305} C_VEL
LIN {X 0,Y 461.082,Z 187.664,A -85,B 0,C 180,E1 -8046.473,E2 -8046.473} C_VEL
LIN {X 0,Y 461.382,Z 183.87,A -85,B 0,C 180,E1 -8049.026,E2 -8049.026} C_VEL
LIN {X 0,Y 461.503,Z 180.108,A -85,B 0,C 180,E1 -8051.738,E2 -8051.738} C_VEL
LIN {X 0,Y 461.133,Z 176.626,A -85,B 0,C 180,E1 -8054.512,E2 -8054.512} C_VEL
LIN {X 0,Y 460.52,Z 172.809,A -85,B 0,C 180,E1 -8057.818,E2 -8057.818} C_VEL
LIN {X 0,Y 460.522,Z 172.622,A -85,B 0,C 180,E1 -8060.136,E2 -8060.136} C_VEL
LIN {X 0,Y 460.474,Z 172.623,A -85,B 0,C 180,E1 -8063.47,E2 -8063.47} C_VEL
LIN {X 0,Y 460.526,Z 172.624,A -85,B 0,C 180,E1 -8066.674,E2 -8066.674} C_VEL
LIN {X 0,Y 460.507,Z 172.618,A -85,B 0,C 180,E1 -8069.759,E2 -8069.759} C_VEL
LIN {X 0,Y 460.568,Z 172.615,A -85,B 0,C 180,E1 -8072.755,E2 -8072.755} C_VEL
LIN {X 0,Y 460.539,Z 172.614,A -85,B 0,C 180,E1 -8075.667,E2 -8075.667} C_VEL
LIN {X 0,Y 460.517,Z 172.621,A -85,B 0,C 180,E1 -8078.577,E2 -8078.577} C_VEL
LIN {X 0,Y 460.586,Z 172.608,A -85,B 0,C 180,E1 -8081.31,E2 -8081.31} C_VEL
LIN {X 0,Y 460.599,Z 172.613,A -85,B 0,C 180,E1 -8084.058,E2 -8084.058} C_VEL
LIN {X 0,Y 460.604,Z 172.609,A -85,B 0,C 180,E1 -8087.665,E2 -8087.665} C_VEL
LIN {X 0,Y 460.623,Z 172.604,A -85,B 0,C 180,E1 -8091.223,E2 -8091.223} C_VEL
LIN {X 0,Y 460.697,Z 172.602,A -85,B 0,C 180,E1 -8093.869,E2 -8093.869} C_VEL
LIN {X 0,Y 460.793,Z 172.585,A -85,B 0,C 180,E1 -8097.377,E2 -8097.377} C_VEL
LIN {X 0,Y 460.846,Z 172.579,A -85,B 0,C 180,E1 -8100,E2 -8100} C_VEL
LIN {X 0,Y 460.794,Z 172.582,A -85,B 0,C 180,E1 -8102.622,E2 -8102.622} C_VEL
LIN {X 0,Y 460.703,Z 172.595,A -85,B 0,C 180,E1 -8106.13,E2 -8106.13} C_VEL
LIN {X 0,Y 460.622,Z 172.604,A -85,B 0,C 180,E1 -8108.776,E2 -8108.776} C_VEL
LIN {X 0,Y 460.607,Z 172.606,A -85,B 0,C 180,E1 -8112.445,E2 -8112.445} C_VEL
LIN {X 0,Y 460.593,Z 172.607,A -85,B 0,C 180,E1 -8115.997,E2 -8115.997} C_VEL
LIN {X 0,Y 460.564,Z 172.616,A -85,B 0,C 180,E1 -8118.902,E2 -8118.902} C_VEL
LIN {X 0,Y 460.509,Z 172.62,A -85,B 0,C 180,E1 -8121.485,E2 -8121.485} C_VEL
LIN {X 0,Y 460.536,Z 172.615,A -85,B 0,C 180,E1 -8124.332,E2 -8124.332} C_VEL
LIN {X 0,Y 460.573,Z 172.613,A -85,B 0,C 180,E1 -8127.243,E2 -8127.243} C_VEL
LIN {X 0,Y 460.52,Z 172.618,A -85,B 0,C 180,E1 -8130.239,E2 -8130.239} C_VEL
LIN {X 0,Y 460.522,Z 172.617,A -85,B 0,C 180,E1 -8133.325,E2 -8133.325} C_VEL
LIN {X 0,Y 460.472,Z 172.629,A -85,B 0,C 180,E1 -8136.529,E2 -8136.529} C_VEL
LIN {X 0,Y 460.569,Z 172.611,A -85,B 0,C 180,E1 -8139.858,E2 -8139.858} C_VEL
LIN {X 0,Y 460.506,Z 172.62,A -85,B 0,C 180,E1 -8142.9,E2 -8142.9} C_VEL
LIN {X 0,Y 460.505,Z 172.62,A -85,B 0,C 180,E1 -8145.83,E2 -8145.83} C_VEL
LIN {X 0,Y 460.525,Z 172.616,A -85,B 0,C 180,E1 -8148.989,E2 -8148.989} C_VEL
LIN {X 0,Y 460.521,Z 172.616,A -85,B 0,C 180,E1 -8151.267,E2 -8151.267} C_VEL
LIN {X 0,Y 460.508,Z 172.62,A -85,B 0,C 180,E1 -8154.555,E2 -8154.555} C_VEL
LIN {X 0,Y 460.528,Z 172.62,A -85,B 0,C 180,E1 -8157.716,E2 -8157.716} C_VEL
LIN {X 0,Y 460.543,Z 172.613,A -85,B 0,C 180,E1 -8160.77,E2 -8160.77} C_VEL
LIN {X 0,Y 460.558,Z 172.619,A -85,B 0,C 180,E1 -8163.735,E2 -8163.735} C_VEL
LIN {X 0,Y 460.542,Z 172.614,A -85,B 0,C 180,E1 -8166.624,E2 -8166.624} C_VEL
LIN {X 0,Y 460.548,Z 172.619,A -85,B 0,C 180,E1 -8169.453,E2 -8169.453} C_VEL
LIN {X 0,Y 460.555,Z 172.616,A -85,B 0,C 180,E1 -8172.23,E2 -8172.23} C_VEL
LIN {X 0,Y 460.564,Z 172.616,A -85,B 0,C 180,E1 -8174.965,E2 -8174.965} C_VEL
LIN {X 0,Y 460.608,Z 172.608,A -85,B 0,C 180,E1 -8178.559,E2 -8178.559} C_VEL
LIN {X 0,Y 460.574,Z 172.614,A -85,B 0,C 180,E1 -8179.222,E2 -8179.222} C_VEL
LIN {X 0,Y 459.919,Z 172.7,A -85,B 0,C 180,E1 -8179.953,E2 -8179.953} C_VEL
LIN {X 0,Y 457.101,Z 173.055,A -85,B 0,C 180,E1 -8181.139,E2 -8181.139} C_VEL
LIN {X 0,Y 454.722,Z 173.349,A -85,B 0,C 180,E1 -8182.096,E2 -8182.096} C_VEL
LIN {X 0,Y 453.711,Z 173.471,A -85,B 0,C 180,E1 -8182.835,E2 -8182.835} C_VEL
LIN {X 0,Y 453.634,Z 173.479,A -85,B 0,C 180,E1 -8183.085,E2 -8183.085} C_VEL
LIN {X 0,Y 453.67,Z 173.474,A -85,B 0,C 180,E1 -8184.667,E2 -8184.667} C_VEL
LIN {X 0,Y 453.762,Z 173.466,A -85,B 0,C 180,E1 -8187.337,E2 -8187.337} C_VEL
LIN {X 0,Y 453.821,Z 173.455,A -85,B 0,C 180,E1 -8190,E2 -8190} C_VEL
LIN {X 0,Y 453.762,Z 173.466,A -85,B 0,C 180,E1 -8192.663,E2 -8192.663} C_VEL
LIN {X 0,Y 453.676,Z 173.474,A -85,B 0,C 180,E1 -8196.225,E2 -8196.225} C_VEL
LIN {X 0,Y 453.589,Z 173.486,A -85,B 0,C 180,E1 -8198.913,E2 -8198.913} C_VEL
LIN {X 0,Y 453.559,Z 173.49,A -85,B 0,C 180,E1 -8202.529,E2 -8202.529} C_VEL
LIN {X 0,Y 453.541,Z 173.492,A -85,B 0,C 180,E1 -8206.196,E2 -8206.196} C_VEL
LIN {X 0,Y 453.516,Z 173.492,A -85,B 0,C 180,E1 -8209.041,E2 -8209.041} C_VEL
LIN {X 0,Y 453.473,Z 173.496,A -85,B 0,C 180,E1 -8211.836,E2 -8211.836} C_VEL
LIN {X 0,Y 453.51,Z 173.492,A -85,B 0,C 180,E1 -8214.734,E2 -8214.734} C_VEL
LIN {X 0,Y 453.534,Z 173.492,A -85,B 0,C 180,E1 -8217.961,E2 -8217.961} C_VEL
LIN {X 0,Y 453.478,Z 173.494,A -85,B 0,C 180,E1 -8220.759,E2 -8220.759} C_VEL
LIN {X 0,Y 453.473,Z 173.501,A -85,B 0,C 180,E1 -8223.912,E2 -8223.912} C_VEL
LIN {X 0,Y 453.466,Z 173.496,A -85,B 0,C 180,E1 -8227.188,E2 -8227.188} C_VEL
LIN {X 0,Y 453.523,Z 173.491,A -85,B 0,C 180,E1 -8229.446,E2 -8229.446} C_VEL
LIN {X 0,Y 453.473,Z 173.5,A -85,B 0,C 180,E1 -8231.935,E2 -8231.935} C_VEL
LIN {X 0,Y 453.481,Z 173.499,A -85,B 0,C 180,E1 -8235.471,E2 -8235.471} C_VEL
LIN {X 0,Y 453.475,Z 173.495,A -85,B 0,C 180,E1 -8238.21,E2 -8238.21} C_VEL
LIN {X 0,Y 453.524,Z 173.489,A -85,B 0,C 180,E1 -8240.788,E2 -8240.788} C_VEL
LIN {X 0,Y 453.451,Z 173.499,A -85,B 0,C 180,E1 -8243.918,E2 -8243.918} C_VEL
LIN {X 0,Y 453.476,Z 173.5,A -85,B 0,C 180,E1 -8247.151,E2 -8247.151} C_VEL
LIN {X 0,Y 453.508,Z 173.49,A -85,B 0,C 180,E1 -8250.271,E2 -8250.271} C_VEL
LIN {X 0,Y 453.503,Z 173.496,A -85,B 0,C 180,E1 -8253.294,E2 -8253.294} C_VEL
LIN {X 0,Y 453.497,Z 173.492,A -85,B 0,C 180,E1 -8256.239,E2 -8256.239} C_VEL
LIN {X 0,Y 453.476,Z 173.499,A -85,B 0,C 180,E1 -8259.118,E2 -8259.118} C_VEL
LIN {X 0,Y 453.505,Z 173.49,A -85,B 0,C 180,E1 -8261.945,E2 -8261.945} C_VEL
LIN {X 0,Y 453.533,Z 173.494,A -85,B 0,C 180,E1 -8264.727,E2 -8264.727} C_VEL
LIN {X 0,Y 453.553,Z 173.488,A -85,B 0,C 180,E1 -8268.379,E2 -8268.379} C_VEL
LIN {X 0,Y 453.646,Z 173.474,A -85,B 0,C 180,E1 -8271.986,E2 -8271.986} C_VEL
LIN {X 0,Y 453.664,Z 173.476,A -85,B 0,C 180,E1 -8274.667,E2 -8274.667} C_VEL
LIN {X 0,Y 453.738,Z 173.461,A -85,B 0,C 180,E1 -8277.337,E2 -8277.337} C_VEL
LIN {X 0,Y 453.817,Z 173.455,A -85,B 0,C 180,E1 -8280,E2 -8280} C_VEL
LIN {X 0,Y 453.737,Z 173.464,A -85,B 0,C 180,E1 -8282.664,E2 -8282.664} C_VEL
LIN {X 0,Y 453.665,Z 173.477,A -85,B 0,C 180,E1 -8286.226,E2 -8286.226} C_VEL
LIN {X 0,Y 453.587,Z 173.48,A -85,B 0,C 180,E1 -8288.914,E2 -8288.914} C_VEL
LIN {X 0,Y 453.559,Z 173.485,A -85,B 0,C 180,E1 -8292.529,E2 -8292.529} C_VEL
LIN {X 0,Y 453.54,Z 173.489,A -85,B 0,C 180,E1 -8296.197,E2 -8296.197} C_VEL
LIN {X 0,Y 453.515,Z 173.49,A -85,B 0,C 180,E1 -8299.041,E2 -8299.041} C_VEL
LIN {X 0,Y 453.472,Z 173.5,A -85,B 0,C 180,E1 -8301.837,E2 -8301.837} C_VEL
LIN {X 0,Y 453.51,Z 173.49,A -85,B 0,C 180,E1 -8304.735,E2 -8304.735} C_VEL
LIN {X 0,Y 453.528,Z 173.489,A -85,B 0,C 180,E1 -8307.96,E2 -8307.96} C_VEL
LIN {X 0,Y 453.463,Z 173.501,A -85,B 0,C 180,E1 -8311.526,E2 -8311.526} C_VEL
LIN {X 0,Y 453.484,Z 173.497,A -85,B 0,C 180,E1 -8314.778,E2 -8314.778} C_VEL
LIN {X 0,Y 453.46,Z 173.501,A -85,B 0,C 180,E1 -8318.313,E2 -8318.313} C_VEL
LIN {X 0,Y 453.491,Z 173.498,A -85,B 0,C 180,E1 -8320.61,E2 -8320.61} C_VEL
LIN {X 0,Y 453.523,Z 173.785,A -85,B 0,C 180,E1 -8321.942,E2 -8321.942} C_VEL
LIN {X 0,Y 454.115,Z 177.674,A -85,B 0,C 180,E1 -8325.391,E2 -8325.391} C_VEL
LIN {X 0,Y 454.486,Z 180.807,A -85,B 0,C 180,E1 -8327.924,E2 -8327.924} C_VEL
LIN {X 0,Y 454.388,Z 184.511,A -85,B 0,C 180,E1 -8330.656,E2 -8330.656} C_VEL
LIN {X 0,Y 454.048,Z 188.789,A -85,B 0,C 180,E1 -8333.6,E2 -8333.6} C_VEL
LIN {X 0,Y 453.737,Z 193.69,A -85,B 0,C 180,E1 -8336.764,E2 -8336.764} C_VEL
LIN {X 0,Y 453.516,Z 197.727,A -85,B 0,C 180,E1 -8339.244,E2 -8339.244} C_VEL
LIN {X 0,Y 453.298,Z 202.883,A -85,B 0,C 180,E1 -8342.282,E2 -8342.282} C_VEL
LIN {X 0,Y 453.086,Z 208.131,A -85,B 0,C 180,E1 -8345.241,E2 -8345.241} C_VEL
LIN {X 0,Y 452.914,Z 214.307,A -85,B 0,C 180,E1 -8348.598,E2 -8348.598} C_VEL
LIN {X 0,Y 452.703,Z 220.611,A -85,B 0,C 180,E1 -8351.911,E2 -8351.911} C_VEL
LIN {X 0,Y 452.659,Z 224.929,A -85,B 0,C 180,E1 -8354.125,E2 -8354.125} C_VEL
LIN {X 0,Y 454.709,Z 236.129,A -85,B 0,C 180,E1 -8354.508,E2 -8354.508} C_VEL
LIN {X 0,Y 456.214,Z 245.714,A -85,B 0,C 180,E1 -8354.933,E2 -8354.933} C_VEL
LIN {X 0,Y 455.949,Z 254.794,A -85,B 0,C 180,E1 -8355.38,E2 -8355.38} C_VEL
LIN {X 0,Y 455.511,Z 263.931,A -85,B 0,C 180,E1 -8355.936,E2 -8355.936} C_VEL
LIN {X 0,Y 455.049,Z 272.932,A -85,B 0,C 180,E1 -8356.605,E2 -8356.605} C_VEL
LIN {X 0,Y 454.675,Z 281.142,A -85,B 0,C 180,E1 -8357.337,E2 -8357.337} C_VEL
LIN {X 0,Y 454.267,Z 289.066,A -85,B 0,C 180,E1 -8358.171,E2 -8358.171} C_VEL
LIN {X 0,Y 453.826,Z 296.288,A -85,B 0,C 180,E1 -8359.065,E2 -8359.065} C_VEL
LIN {X 0,Y 453.534,Z 302.494,A -85,B 0,C 180,E1 -8359.96,E2 -8359.96} C_VEL
LIN {X 0,Y 453.199,Z 309.034,A -85,B 0,C 180,E1 -8361.079,E2 -8361.079} C_VEL
LIN {X 0,Y 452.927,Z 313.536,A -85,B 0,C 180,E1 -8361.972,E2 -8361.972} C_VEL
LIN {X 0,Y 452.739,Z 318.6,A -85,B 0,C 180,E1 -8363.191,E2 -8363.191} C_VEL
LIN {X 0,Y 452.619,Z 323.354,A -85,B 0,C 180,E1 -8364.654,E2 -8364.654} C_VEL
LIN {X 0,Y 452.505,Z 325.718,A -85,B 0,C 180,E1 -8365.546,E2 -8365.546} C_VEL
LIN {X 0,Y 452.492,Z 327.516,A -85,B 0,C 180,E1 -8366.438,E2 -8366.438} C_VEL
LIN {X 0,Y 452.433,Z 329.958,A -85,B 0,C 180,E1 -8368.22,E2 -8368.22} C_VEL
LIN {X 0,Y 452.403,Z 330.545,A -85,B 0,C 180,E1 -8369.11,E2 -8369.11} C_VEL
LIN {X 0,Y 452.403,Z 330.545,A -85,B 0,C 180,E1 -8370.89,E2 -8370.89} C_VEL
LIN {X 0,Y 452.433,Z 329.958,A -85,B 0,C 180,E1 -8371.78,E2 -8371.78} C_VEL
LIN {X 0,Y 452.492,Z 327.516,A -85,B 0,C 180,E1 -8373.562,E2 -8373.562} C_VEL
LIN {X 0,Y 452.567,Z 324.57,A -85,B 0,C 180,E1 -8374.9,E2 -8374.9} C_VEL
LIN {X 0,Y 452.663,Z 320.582,A -85,B 0,C 180,E1 -8376.239,E2 -8376.239} C_VEL
LIN {X 0,Y 452.831,Z 315.452,A -85,B 0,C 180,E1 -8377.58,E2 -8377.58} C_VEL
LIN {X 0,Y 453.115,Z 310.189,A -85,B 0,C 180,E1 -8378.698,E2 -8378.698} C_VEL
LIN {X 0,Y 453.458,Z 303.871,A -85,B 0,C 180,E1 -8379.816,E2 -8379.816} C_VEL
LIN {X 0,Y 453.72,Z 297.915,A -85,B 0,C 180,E1 -8380.712,E2 -8380.712} C_VEL
LIN {X 0,Y 454.126,Z 290.985,A -85,B 0,C 180,E1 -8381.606,E2 -8381.606} C_VEL
LIN {X 0,Y 454.587,Z 282.801,A -85,B 0,C 180,E1 -8382.5,E2 -8382.5} C_VEL
LIN {X 0,Y 454.912,Z 275.802,A -85,B 0,C 180,E1 -8383.158,E2 -8383.158} C_VEL
LIN {X 0,Y 455.414,Z 265.563,A -85,B 0,C 180,E1 -8383.953,E2 -8383.953} C_VEL
LIN {X 0,Y 455.871,Z 255.801,A -85,B 0,C 180,E1 -8384.565,E2 -8384.565} C_VEL
LIN {X 0,Y 456.23,Z 247.004,A -85,B 0,C 180,E1 -8385.01,E2 -8385.01} C_VEL
LIN {X 0,Y 454.912,Z 237.277,A -85,B 0,C 180,E1 -8385.447,E2 -8385.447} C_VEL
LIN {X 0,Y 452.899,Z 226.739,A -85,B 0,C 180,E1 -8385.822,E2 -8385.822} C_VEL
LIN {X 0,Y 452.655,Z 224.938,A -85,B 0,C 180,E1 -8385.871,E2 -8385.871} C_VEL
LIN {X 0,Y 452.767,Z 218.811,A -85,B 0,C 180,E1 -8389.024,E2 -8389.024} C_VEL
LIN {X 0,Y 452.939,Z 213.439,A -85,B 0,C 180,E1 -8391.863,E2 -8391.863} C_VEL
LIN {X 0,Y 453.086,Z 208.118,A -85,B 0,C 180,E1 -8394.759,E2 -8394.759} C_VEL
LIN {X 0,Y 453.321,Z 202.548,A -85,B 0,C 180,E1 -8397.908,E2 -8397.908} C_VEL
LIN {X 0,Y 453.526,Z 197.711,A -85,B 0,C 180,E1 -8400.755,E2 -8400.755} C_VEL
LIN {X 0,Y 453.771,Z 192.643,A -85,B 0,C 180,E1 -8403.887,E2 -8403.887} C_VEL
LIN {X 0,Y 454.128,Z 187.7,A -85,B 0,C 180,E1 -8407.124,E2 -8407.124} C_VEL
LIN {X 0,Y 454.384,Z 184.473,A -85,B 0,C 180,E1 -8409.356,E2 -8409.356} C_VEL
LIN {X 0,Y 454.488,Z 180.806,A -85,B 0,C 180,E1 -8412.076,E2 -8412.076} C_VEL
LIN {X 0,Y 454.118,Z 177.672,A -85,B 0,C 180,E1 -8414.61,E2 -8414.61} C_VEL
LIN {X 0,Y 453.483,Z 173.625,A -85,B 0,C 180,E1 -8418.209,E2 -8418.209} C_VEL
LIN {X 0,Y 453.488,Z 173.5,A -85,B 0,C 180,E1 -8420.793,E2 -8420.793} C_VEL
LIN {X 0,Y 453.451,Z 173.498,A -85,B 0,C 180,E1 -8423.916,E2 -8423.916} C_VEL
LIN {X 0,Y 453.48,Z 173.495,A -85,B 0,C 180,E1 -8427.15,E2 -8427.15} C_VEL
LIN {X 0,Y 453.47,Z 173.498,A -85,B 0,C 180,E1 -8430.268,E2 -8430.268} C_VEL
LIN {X 0,Y 453.502,Z 173.491,A -85,B 0,C 180,E1 -8433.293,E2 -8433.293} C_VEL
LIN {X 0,Y 453.5,Z 173.497,A -85,B 0,C 180,E1 -8436.238,E2 -8436.238} C_VEL
LIN {X 0,Y 453.478,Z 173.494,A -85,B 0,C 180,E1 -8439.117,E2 -8439.117} C_VEL
LIN {X 0,Y 453.506,Z 173.494,A -85,B 0,C 180,E1 -8441.944,E2 -8441.944} C_VEL
LIN {X 0,Y 453.535,Z 173.488,A -85,B 0,C 180,E1 -8444.726,E2 -8444.726} C_VEL
LIN {X 0,Y 453.554,Z 173.487,A -85,B 0,C 180,E1 -8448.378,E2 -8448.378} C_VEL
LIN {X 0,Y 453.647,Z 173.48,A -85,B 0,C 180,E1 -8451.985,E2 -8451.985} C_VEL
LIN {X 0,Y 453.662,Z 173.471,A -85,B 0,C 180,E1 -8454.666,E2 -8454.666} C_VEL
LIN {X 0,Y 453.737,Z 173.464,A -85,B 0,C 180,E1 -8457.336,E2 -8457.336} C_VEL
LIN {X 0,Y 453.817,Z 173.455,A -85,B 0,C 180,E1 -8460,E2 -8460} C_VEL
LIN {X 0,Y 453.738,Z 173.461,A -85,B 0,C 180,E1 -8462.663,E2 -8462.663} C_VEL
LIN {X 0,Y 453.67,Z 173.47,A -85,B 0,C 180,E1 -8466.225,E2 -8466.225} C_VEL
LIN {X 0,Y 453.586,Z 173.482,A -85,B 0,C 180,E1 -8468.913,E2 -8468.913} C_VEL
LIN {X 0,Y 453.557,Z 173.484,A -85,B 0,C 180,E1 -8472.528,E2 -8472.528} C_VEL
LIN {X 0,Y 453.538,Z 173.486,A -85,B 0,C 180,E1 -8476.196,E2 -8476.196} C_VEL
LIN {X 0,Y 453.514,Z 173.496,A -85,B 0,C 180,E1 -8479.041,E2 -8479.041} C_VEL
LIN {X 0,Y 453.47,Z 173.495,A -85,B 0,C 180,E1 -8481.836,E2 -8481.836} C_VEL
LIN {X 0,Y 453.507,Z 173.495,A -85,B 0,C 180,E1 -8484.734,E2 -8484.734} C_VEL
LIN {X 0,Y 453.532,Z 173.487,A -85,B 0,C 180,E1 -8487.961,E2 -8487.961} C_VEL
LIN {X 0,Y 453.477,Z 173.502,A -85,B 0,C 180,E1 -8490.759,E2 -8490.759} C_VEL
LIN {X 0,Y 453.471,Z 173.495,A -85,B 0,C 180,E1 -8493.913,E2 -8493.913} C_VEL
LIN {X 0,Y 453.465,Z 173.496,A -85,B 0,C 180,E1 -8497.188,E2 -8497.188} C_VEL
LIN {X 0,Y 453.525,Z 173.488,A -85,B 0,C 180,E1 -8499.445,E2 -8499.445} C_VEL
LIN {X 0,Y 453.456,Z 173.498,A -85,B 0,C 180,E1 -8502.995,E2 -8502.995} C_VEL
LIN {X 0,Y 453.46,Z 173.497,A -85,B 0,C 180,E1 -8505.779,E2 -8505.779} C_VEL
LIN {X 0,Y 453.473,Z 173.502,A -85,B 0,C 180,E1 -8508.209,E2 -8508.209} C_VEL
LIN {X 0,Y 453.51,Z 173.491,A -85,B 0,C 180,E1 -8510.79,E2 -8510.79} C_VEL
LIN {X 0,Y 453.452,Z 173.502,A -85,B 0,C 180,E1 -8513.918,E2 -8513.918} C_VEL
LIN {X 0,Y 453.478,Z 173.494,A -85,B 0,C 180,E1 -8517.151,E2 -8517.151} C_VEL
LIN {X 0,Y 453.509,Z 173.493,A -85,B 0,C 180,E1 -8520.271,E2 -8520.271} C_VEL
LIN {X 0,Y 453.504,Z 173.492,A -85,B 0,C 180,E1 -8523.294,E2 -8523.294} C_VEL
LIN {X 0,Y 453.499,Z 173.493,A -85,B 0,C 180,E1 -8526.239,E2 -8526.239} C_VEL
LIN {X 0,Y 453.479,Z 173.495,A -85,B 0,C 180,E1 -8529.118,E2 -8529.118} C_VEL
LIN {X 0,Y 453.508,Z 173.496,A -85,B 0,C 180,E1 -8531.945,E2 -8531.945} C_VEL
LIN {X 0,Y 453.538,Z 173.49,A -85,B 0,C 180,E1 -8534.726,E2 -8534.726} C_VEL
LIN {X 0,Y 453.556,Z 173.486,A -85,B 0,C 180,E1 -8538.379,E2 -8538.379} C_VEL
LIN {X 0,Y 453.648,Z 173.477,A -85,B 0,C 180,E1 -8541.985,E2 -8541.985} C_VEL
LIN {X 0,Y 453.634,Z 173.479,A -85,B 0,C 180,E1 -8543.085,E2 -8543.085} C_VEL
LIN {X 0,Y 452.949,Z 173.565,A -85,B 0,C 180,E1 -8543.826,E2 -8543.826} C_VEL
LIN {X 0,Y 449.999,Z 173.934,A -85,B 0,C 180,E1 -8545.027,E2 -8545.027} C_VEL
LIN {X 0,Y 447.576,Z 174.234,A -85,B 0,C 180,E1 -8545.997,E2 -8545.997} C_VEL
LIN {X 0,Y 446.639,Z 174.351,A -85,B 0,C 180,E1 -8546.747,E2 -8546.747} C_VEL
LIN {X 0,Y 446.619,Z 174.353,A -85,B 0,C 180,E1 -8547.001,E2 -8547.001} C_VEL
LIN {X 0,Y 446.791,Z 174.331,A -85,B 0,C 180,E1 -8550,E2 -8550} C_VEL
LIN {X 0,Y 446.706,Z 174.344,A -85,B 0,C 180,E1 -8552.705,E2 -8552.705} C_VEL
LIN {X 0,Y 446.645,Z 174.35,A -85,B 0,C 180,E1 -8556.324,E2 -8556.324} C_VEL
LIN {X 0,Y 446.535,Z 174.364,A -85,B 0,C 180,E1 -8559.055,E2 -8559.055} C_VEL
LIN {X 0,Y 446.518,Z 174.368,A -85,B 0,C 180,E1 -8562.73,E2 -8562.73} C_VEL
LIN {X 0,Y 446.492,Z 174.37,A -85,B 0,C 180,E1 -8566.228,E2 -8566.228} C_VEL
LIN {X 0,Y 446.465,Z 174.368,A -85,B 0,C 180,E1 -8569.303,E2 -8569.303} C_VEL
LIN {X 0,Y 446.415,Z 174.379,A -85,B 0,C 180,E1 -8572.199,E2 -8572.199} C_VEL
LIN {X 0,Y 446.453,Z 174.369,A -85,B 0,C 180,E1 -8575.152,E2 -8575.152} C_VEL
LIN {X 0,Y 446.48,Z 174.373,A -85,B 0,C 180,E1 -8578.179,E2 -8578.179} C_VEL
LIN {X 0,Y 446.415,Z 174.374,A -85,B 0,C 180,E1 -8581.3,E2 -8581.3} C_VEL
LIN {X 0,Y 446.425,Z 174.374,A -85,B 0,C 180,E1 -8584.523,E2 -8584.523} C_VEL
LIN {X 0,Y 446.43,Z 174.376,A -85,B 0,C 180,E1 -8588.083,E2 -8588.083} C_VEL
LIN {X 0,Y 446.437,Z 174.371,A -85,B 0,C 180,E1 -8590.92,E2 -8590.92} C_VEL
LIN {X 0,Y 446.395,Z 174.382,A -85,B 0,C 180,E1 -8593.846,E2 -8593.846} C_VEL
LIN {X 0,Y 446.393,Z 174.376,A -85,B 0,C 180,E1 -8596.403,E2 -8596.403} C_VEL
LIN {X 0,Y 446.462,Z 174.372,A -85,B 0,C 180,E1 -8599.805,E2 -8599.805} C_VEL
LIN {X 0,Y 446.426,Z 174.373,A -85,B 0,C 180,E1 -8602.124,E2 -8602.124} C_VEL
LIN {X 0,Y 446.424,Z 174.378,A -85,B 0,C 180,E1 -8605.477,E2 -8605.477} C_VEL
LIN {X 0,Y 446.413,Z 174.375,A -85,B 0,C 180,E1 -8608.7,E2 -8608.7} C_VEL
LIN {X 0,Y 446.478,Z 174.366,A -85,B 0,C 180,E1 -8611.822,E2 -8611.822} C_VEL
LIN {X 0,Y 446.451,Z 174.374,A -85,B 0,C 180,E1 -8614.848,E2 -8614.848} C_VEL
LIN {X 0,Y 446.441,Z 174.371,A -85,B 0,C 180,E1 -8618.245,E2 -8618.245} C_VEL
LIN {X 0,Y 446.451,Z 174.369,A -85,B 0,C 180,E1 -8621.649,E2 -8621.649} C_VEL
LIN {X 0,Y 446.501,Z 174.367,A -85,B 0,C 180,E1 -8624.48,E2 -8624.48} C_VEL
LIN {X 0,Y 446.511,Z 174.364,A -85,B 0,C 180,E1 -8628.193,E2 -8628.193} C_VEL
LIN {X 0,Y 446.594,Z 174.352,A -85,B 0,C 180,E1 -8631.858,E2 -8631.858} C_VEL
LIN {X 0,Y 446.638,Z 174.352,A -85,B 0,C 180,E1 -8634.583,E2 -8634.583} C_VEL
LIN {X 0,Y 446.658,Z 174.349,A -85,B 0,C 180,E1 -8638.197,E2 -8638.197} C_VEL
LIN {X 0,Y 446.787,Z 174.331,A -85,B 0,C 180,E1 -8640,E2 -8640} C_VEL
LIN {X 0,Y 446.685,Z 174.342,A -85,B 0,C 180,E1 -8642.706,E2 -8642.706} C_VEL
LIN {X 0,Y 446.635,Z 174.351,A -85,B 0,C 180,E1 -8646.324,E2 -8646.324} C_VEL
LIN {X 0,Y 446.533,Z 174.359,A -85,B 0,C 180,E1 -8649.056,E2 -8649.056} C_VEL
LIN {X 0,Y 446.517,Z 174.361,A -85,B 0,C 180,E1 -8652.73,E2 -8652.73} C_VEL
LIN {X 0,Y 446.491,Z 174.367,A -85,B 0,C 180,E1 -8656.228,E2 -8656.228} C_VEL
LIN {X 0,Y 446.465,Z 174.37,A -85,B 0,C 180,E1 -8659.304,E2 -8659.304} C_VEL
LIN {X 0,Y 446.414,Z 174.375,A -85,B 0,C 180,E1 -8662.2,E2 -8662.2} C_VEL
LIN {X 0,Y 446.454,Z 174.371,A -85,B 0,C 180,E1 -8665.153,E2 -8665.153} C_VEL
LIN {X 0,Y 446.481,Z 174.366,A -85,B 0,C 180,E1 -8668.179,E2 -8668.179} C_VEL
LIN {X 0,Y 446.416,Z 174.376,A -85,B 0,C 180,E1 -8671.776,E2 -8671.776} C_VEL
LIN {X 0,Y 446.426,Z 174.375,A -85,B 0,C 180,E1 -8674.524,E2 -8674.524} C_VEL
LIN {X 0,Y 446.412,Z 174.379,A -85,B 0,C 180,E1 -8678.08,E2 -8678.08} C_VEL
LIN {X 0,Y 446.422,Z 174.38,A -85,B 0,C 180,E1 -8680.918,E2 -8680.918} C_VEL
LIN {X 0,Y 446.43,Z 174.431,A -85,B 0,C 180,E1 -8681.391,E2 -8681.391} C_VEL
LIN {X 0,Y 447.039,Z 178.354,A -85,B 0,C 180,E1 -8684.973,E2 -8684.973} C_VEL
LIN {X 0,Y 447.444,Z 181.511,A -85,B 0,C 180,E1 -8687.581,E2 -8687.581} C_VEL
LIN {X 0,Y 447.411,Z 184.541,A -85,B 0,C 180,E1 -8689.907,E2 -8689.907} C_VEL
LIN {X 0,Y 447.177,Z 187.744,A -85,B 0,C 180,E1 -8692.198,E2 -8692.198} C_VEL
LIN {X 0,Y 446.818,Z 192.666,A -85,B 0,C 180,E1 -8695.512,E2 -8695.512} C_VEL
LIN {X 0,Y 446.503,Z 197.692,A -85,B 0,C 180,E1 -8698.707,E2 -8698.707} C_VEL
LIN {X 0,Y 446.265,Z 202.942,A -85,B 0,C 180,E1 -8701.875,E2 -8701.875} C_VEL
LIN {X 0,Y 446.031,Z 208.035,A -85,B 0,C 180,E1 -8704.822,E2 -8704.822} C_VEL
LIN {X 0,Y 445.839,Z 214.557,A -85,B 0,C 180,E1 -8708.443,E2 -8708.443} C_VEL
LIN {X 0,Y 445.631,Z 220.456,A -85,B 0,C 180,E1 -8711.614,E2 -8711.614} C_VEL
